	ELSIF ENABLE THEN
		IF trig_tmp OR trig_stored THEN (* manueller, automatischer oder externer Trigger *)
			trig_stored := FALSE;
			X.ADD_COM := 03; (* ADD DATA *)
			SAVE_DATA.TRIG_CNT := SAVE_DATA.TRIG_CNT + UDINT#1;
			SAVE_DATA.TRIG_CNT_TOTAL  := SAVE_DATA.TRIG_CNT_TOTAL + UDINT#1;
			(* ---------------- Debug-Message -----------------------*)
			(*IF _debug_enable THEN
				LOG_CL.NEW_MSG := 'FILE_XML1 - Trig: [~2]';
				LOG_CL.PRINTF[2] := DT_TO_STRING(DTI);
				LOG_MSG();
			END_IF;*)
			(* -----------------------------------------------------------------*)
		ELSE
			X.ADD_COM := 04;	(* ADD DATA REQ *)
		END_IF;
	END_IF;

END_CASE;
X.ADD_DATA_REQ := FALSE; (* externe Anforderung rücksetzen *)

(* ##################################### *)

CASE step_2 OF

00:	aw_ton(IN:= idx > 0 AND aw_enable , PT:= AUTO_CLOSE); (* AutoWrite Timer *)
	IF aw_ton.Q THEN (* Zeitgesteuertes Datenschreiben *)
		aw_aktiv := TRUE;
		step_2 := 10; (* Daten schreiben *)
		(* ---------------- Debug-Message -----------------------*)
		(*IF _debug_enable THEN
			LOG_CL.NEW_MSG := 'FILE_XML2 - AutoWrite: [~2]';
			LOG_CL.PRINTF[2] := DT_TO_STRING(DTI);
			LOG_MSG();
		END_IF;*)
		(* -----------------------------------------------------------------*)

	ELSIF idx + 256 > SIZEOF(PT.BUFFER) THEN (* Platz für Element vorhanden ? *)
		step_2 := 10; (* Daten schreiben *)
	ELSE
		wd_ton(IN:= FALSE, PT:= wd_time);
		wd_ton(IN:= TRUE);
		WHILE X.UCB.BUF_COUNT > 0 AND step_2 = 0 AND wd_ton.Q = FALSE DO

			X.UCB.D_MODE := 10;
			UCB(DATA:=X.UCB); (* Element lesen , aber noch nicht entfernen *)

			IF X.UCB.D_HEAD > WORD#16#F000 THEN (* F301 oder F201 *)
				X.UCB.D_MODE := 11;
				UCB(DATA:=X.UCB); (* Element entfernen *)

				FSD.MODE := WORD_TO_BYTE(SHR(SHL(X.UCB.D_HEAD,4),12)); (* 0X00 -> 000X = 3 create + write / 2 open + write *)
				FSD.OFFSET := UDINT#0; (* Start bei Dateianfang *)
				FSD.FILENAME := X.UCB.D_STRING; (* Dateiname *)
				PT.SIZE := UINT#0;
				SAVE_DATA.FN_REM := FSD.FILENAME; (* aktuellen Dateinamen remanent sichern *)

				IF FSD.MODE = BYTE#3 THEN	(* Datei neu anlegen -> dann zähler reset *)
					SAVE_DATA.TRIG_CNT := UDINT#0;
				END_IF;

				X.NEW_FILE := FSD.FILENAME;
				X.NEW_FILE_SIZE := UDINT#0;
				X.NEW_FILE_RTRIG := FALSE;
				step_2 := 20;

				(* Headerdaten schreiben *)
				IF FSD.MODE = BYTE#3 THEN
					str := '<?xml version="1.0" encoding="UTF-8"?><table>';
					_STRING_TO_BUFFER(STR:=str, POS:=idx, PT:=ADR(PT.BUFFER), SIZE:=SIZEOF(PT.BUFFER));
					idx := LEN(str);
					X.NEW_FILE_SIZE := total_bytes + INT_TO_UDINT(idx);
				END_IF;

				(* ---------------- Debug-Message -----------------------*)
				(*IF _debug_enable THEN
					LOG_CL.NEW_MSG := 'FILE_XML2 - Create: Mode [~1] , [~2]';
					LOG_CL.PRINTF[2] := DT_TO_STRING(DTI);
					LOG_CL.PRINTF[1] := BYTE_TO_STRING(FSD.MODE);
					LOG_MSG();
				END_IF;*)
				(* -----------------------------------------------------------------*)

			ELSIF X.UCB.D_HEAD = WORD#16#EE00 THEN (* LOG_STOP Command *)
				X.UCB.D_MODE := 11;
				UCB(DATA:=X.UCB); (* Element entfernen *)

				str := '</table>';
				_STRING_TO_BUFFER(STR:=str, POS:=idx, PT:=ADR(PT.BUFFER), SIZE:=SIZEOF(PT.BUFFER));
				idx := idx + LEN(str);
				log_stop := TRUE;
				step_2 := 10; (* Daten schreiben *)

			ELSE
				X.UCB.D_MODE := 11;
				UCB(DATA:=X.UCB); (* Element entfernen *)
				(* ---------------- Debug-Message -----------------------*)
				(*IF _debug_enable THEN
					LOG_CL.NEW_MSG := 'FILE_XML2 - BUF: TXT [~1],Pos [~2], [~3]';
					LOG_CL.PRINTF[1] := X.UCB.D_STRING;
					LOG_CL.PRINTF[2] := INT_TO_STRING(idx);
					LOG_CL.PRINTF[3] := DT_TO_STRING(DTI);
					LOG_MSG();
				END_IF;*)
				(* -----------------------------------------------------------------*)

				IF log_state = USINT#0 THEN
					str := '<row><entry>';
				ELSE
					str := '<entry>';
				END_IF;

				_STRING_TO_BUFFER(STR:=str, POS:=idx, PT:=ADR(PT.BUFFER), SIZE:=SIZEOF(PT.BUFFER));
				idx := idx + LEN(str);
				log_state := log_state + USINT#1;

				_STRING_TO_BUFFER(STR:=X.UCB.D_STRING, POS:=idx, PT:=ADR(PT.BUFFER), SIZE:=SIZEOF(PT.BUFFER));
				idx := idx + LEN(X.UCB.D_STRING);

				n := n + USINT#1;
				IF n >= X.ID_MAX THEN
					n := USINT#0;
					str := '</entry></row>';
					log_state := USINT#0;
				ELSE
					str := '</entry>';
				END_IF;
				_STRING_TO_BUFFER(STR:=str, POS:=idx, PT:=ADR(PT.BUFFER), SIZE:=SIZEOF(PT.BUFFER));
				idx := idx + LEN(str);
				X.NEW_FILE_SIZE := total_bytes + INT_TO_UDINT(idx);
			END_IF;
			wd_ton();
		END_WHILE;
	END_IF;

10:	IF idx > 0 THEN (* Daten schreiben *)
		FSD.MODE := BYTE#2; (* File_Open_Exist + File_Write *)
		FSD.OFFSET := UDINT#4294967294; (* 16#FFFF_FFFE ->Spezialcode: Daten automatisch an Dateiende anhängen *)
		PT.SIZE := INT_TO_UINT(idx); (* Datenlänge eintragen *)
		idx := 0;
		(* ---------------- Debug-Message -----------------------*)
		(*IF _debug_enable THEN
			LOG_CL.NEW_MSG := 'FILE_XML2 - WriteData: Mode [~3] Size [~1] , [~2]';
			LOG_CL.PRINTF[1] := UINT_TO_STRING(PT.SIZE);
			LOG_CL.PRINTF[2] := DT_TO_STRING(DTI);
			LOG_CL.PRINTF[3] := BYTE_TO_STRING(FSD.MODE);
			LOG_MSG();
		END_IF;*)
		(* -----------------------------------------------------------------*)
	END_IF;
	step_2 := 20;

20:	IF FSD.MODE = BYTE#0 THEN
		total_bytes := FSD.FILE_SIZE;
		X.NEW_FILE_SIZE := total_bytes + INT_TO_UDINT(idx);
		IF log_stop OR aw_aktiv THEN
			aw_aktiv := FALSE;
			FSD.MODE := BYTE#5; (* Datei schliessen *)
			(* ---------------- Debug-Message -----------------------*)
			(*IF _debug_enable THEN
				LOG_CL.NEW_MSG := 'FILE_XML2 - Close: [~2]';
				LOG_CL.PRINTF[2] := DT_TO_STRING(DTI);
				LOG_MSG();
			END_IF;*)
			(* -----------------------------------------------------------------*)
		END_IF;
		step_2 := 30;
	END_IF;

30:	IF FSD.MODE = BYTE#0 THEN (* Datei schliessen beendet *)
		IF log_stop THEN
			X.NEW_FILE_RTRIG := TRUE;
			log_stop := FALSE;
			SAVE_DATA.FN_REM := ''; (* remanenten Dateinamen löschen *)
		END_IF;
		step_2 := 00;
	END_IF;

END_CASE;

FS(FSD:=FSD,PT:=PT); (* FILE_SERVER *)
ERROR_C := BYTE_TO_DWORD(FSD.ERROR);
ERROR_T := SEL(FSD.ERROR > BYTE#0,BYTE#0,BYTE#1);

X.NEW_FILE_SIZE := total_bytes + INT_TO_UDINT(idx);
trig_m_last := TRIG_M;

(* revision history
ks	25. july. 2011	rev 1.0
	original version

ks	16. apr. 2012	rev 1.1
	neuer überarbeiteter Code für automatisches File-open/close
*)
END_FUNCTION_BLOCK

(* POU DLOG_MYSQL_DEMO, CFC *)
PROGRAM DLOG_MYSQL_DEMO
VAR
	cur_dt: DT;
	enable: BOOL := TRUE;
	trig_t : TIME := T#5s;
	trig_m : BOOL;
	error_c: DWORD;
	error_t: BYTE;

	x1 : DLOG_DT;
	x2 : DLOG_REAL;
	x3 : DLOG_DINT;
	x4 : DLOG_BOOL;
	x5 : DLOG_STRING;
	x : DLOG_DATA;
	mysql_info : MYSQL_INFO;

	RTC_2 : RTC_2;
	GEN_SIN_1: GEN_SIN;
	COUNT_DR : COUNT_DR;

	DLOG_STORE_MYSQL : DLOG_STORE_MYSQL;
	(*url : STRING := 'myuser:mypassword@127.0.0.1';*)
	url : STRING(STRING_LENGTH) := 'myuser:mypassword@192.168.178.21';
	db_name : STRING(64) := 'oscat_db';
	tb_name : STRING(64) := 'oscat_tb';
	auto_delete : UDINT := 0;
	timeout : TIME := t#10s;

END_VAR
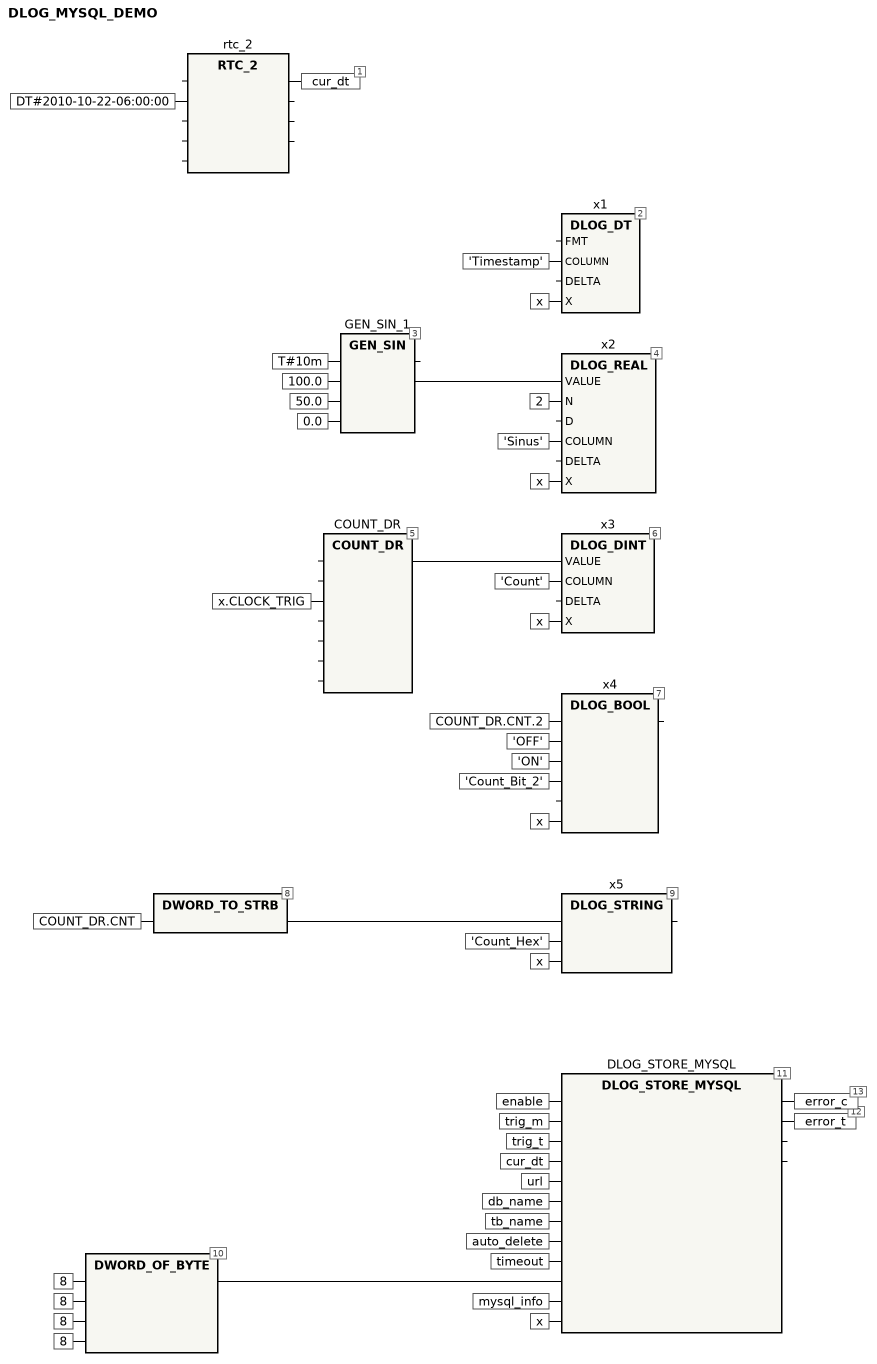
_CFC_ (* Continuous Function Chart, elements in execution order *)
#0 rtc_2:RTC_2(-, DT#2010-10-22-06:00:00, -, -, -)
#1 cur_dt <= #0.out 1
#2 x1:DLOG_DT(FMT: -, COLUMN: 'Timestamp', DELTA: -, X: x)
#3 GEN_SIN_1:GEN_SIN(T#10m, 100.0, 50.0, 0.0)
#4 x2:DLOG_REAL(VALUE: #3.out 2, N: 2, D: -, COLUMN: 'Sinus', DELTA: -, X: x)
#5 COUNT_DR:COUNT_DR(-, -, x.CLOCK_TRIG, -, -, -, -)
#6 x3:DLOG_DINT(VALUE: #5, COLUMN: 'Count', DELTA: -, X: x)
#7 x4:DLOG_BOOL(COUNT_DR.CNT.2, 'OFF', 'ON', 'Count_Bit_2', -, x)
#8 DWORD_TO_STRB(COUNT_DR.CNT)
#9 x5:DLOG_STRING(#8, 'Count_Hex', x)
#10 DWORD_OF_BYTE(8, 8, 8, 8)
#11 DLOG_STORE_MYSQL:DLOG_STORE_MYSQL(enable, trig_m, trig_t, cur_dt, url, db_name, tb_name, auto_delete, timeout, #10, mysql_info, x)
#12 error_t <= #11.out 2
#13 error_c <= #11.out 1
_END_CFC_
END_PROGRAM

(* POU DLOG_STORE_MYSQL, ST *)
FUNCTION_BLOCK DLOG_STORE_MYSQL
VAR_IN_OUT
	SQL_INFO : MYSQL_INFO;
	X : DLOG_DATA;
END_VAR
VAR_INPUT
	ENABLE : BOOL;
	TRIG_M : BOOL;
	TRIG_T : TIME;
	DTI : DT;
	URL : STRING(STRING_LENGTH);
	DB_NAME : STRING(64);
	TB_NAME : STRING(64);
	AUTO_DELETE : UDINT;
	TIMEOUT : TIME;
	DNS_IP4 : DWORD;
END_VAR
VAR_OUTPUT
	ERROR_C : DWORD;
	ERROR_T : BYTE;
END_VAR
VAR
	UCB : UNI_CIRCULAR_BUFFER;
	MYSQL_CONTROL: MYSQL_CONTROL;
	trig_auto : BOOL;
	trig_tmp : BOOL;
	trig_m_last : BOOL;
	dti_last : DT := DT#2070-02-06-06:28:15;
	enable_last : BOOL;
	step : INT;
	idx : INT;
	n : USINT;
	snd_text : STRING(STRING_LENGTH);
	snd_size : INT;
	sql_command : BYTE;
	next_step : INT;
	i1 : INT;
	i2 : INT;
	com: MYSQL_COM;
	del_dt : UDINT;
	del_start : BOOL;
	run : BOOL;

	(*
	LOG_MSG : LOG_MSG;
	_debug_enable : BOOL := TRUE;
	*)
END_VAR

(*
version 1.0		20. apr. 2012
programmer		ks
tested by		ks

DLOG_STORE_MYSQL der Baustein schreibt die DLOG Parameter in eine MySQL Datenbank
*)
X.DTI := DTI; (* Datum / Zeit eintragen *)
X.CLOCK_TRIG := DTI <> dti_last;
dti_last := DTI;
trig_auto := FALSE;
IF X.CLOCK_TRIG THEN (* Impuls in jeder Sekunde *)
	del_start := DT_TO_UDINT(DTI) - del_dt > AUTO_DELETE AND AUTO_DELETE > UDINT#0;
	IF TRIG_T >= T#1000ms THEN (* automatischer Trigger *)
		trig_auto := DT_TO_UDINT(DTI) MOD (TIME_TO_UDINT(TRIG_T) / UDINT#1000) = UDINT#0;
	END_IF;
END_IF;
X.ADD_COM := 00;

CASE step OF

00:	IF ENABLE AND enable_last = FALSE THEN
		COM.SQL_URL := URL;
		COM.TIMEOUT := TIMEOUT;
		COM.DNS_IP4 := DNS_IP4;
		COM.SQL_CON := TRUE;

		X.UCB.D_MODE := 99; (* Buffer reset - Alles löschen *)
		UCB(DATA:=X.UCB);

		X.ID_MAX := USINT#00;
		X.STORE_TYPE := BYTE#5; (* MySQL-Modus *)
		X.ADD_COM := 01; (* ADD INFO *)

		step := 05;
	END_IF;

05:	X.ADD_COM := 02; (* ADD HEADER *)
	step := 10;

10:	IF SQL_INFO.SQL_CONNECTED THEN
		sql_command := BYTE#3; (* CREATE DATABASE IF NOT EXISTS `db_name` *)
		snd_text :=  CONCAT('CREATE DATABASE IF NOT EXISTS `' ,DB_NAME);
		snd_text :=  CONCAT(snd_text, '`');
		next_step := 20;
	END_IF;

20:	sql_command := BYTE#2; (* 0x02 COM_INIT_DB mysql_select_db *)
	snd_text := DB_NAME;
	next_step := 30;

30:	(* CREATE TABLE IF NOT EXISTS tb_name (Timestamp TIMESTAMP NULL DEFAULT CURRENT_TIMESTAMP, n1,n2) *)
	sql_command := BYTE#0;
	idx := 5;
	n := USINT#0;
	WHILE sql_command = BYTE#0 DO
		IF n = USINT#0 THEN
			snd_text := CONCAT('CREATE TABLE IF NOT EXISTS `', TB_NAME);
			snd_text := CONCAT(snd_text,'` (`ID` BIGINT NOT NULL AUTO_INCREMENT PRIMARY KEY ,');
			snd_text := CONCAT(snd_text,' store_timestamp TIMESTAMP NULL DEFAULT CURRENT_TIMESTAMP');
		ELSIF n <= X.ID_MAX THEN
			X.UCB.D_MODE := 12; (* Element lesen und löschen *)
			UCB(DATA:=X.UCB);
			snd_text := CONCAT(', `',X.UCB.D_STRING);
			CASE WORD_TO_INT(SHR(X.UCB.D_HEAD,8)) OF
			02:	snd_text := CONCAT(snd_text, '` FLOAT'); (* REAL *)
			06:	snd_text := CONCAT(snd_text, '` BOOL'); (* BOOL *)
			08:	snd_text := CONCAT(snd_text, '` INT'); (* DINT *)
			13:	snd_text := CONCAT(snd_text, '` DATETIME'); (* DT *)
			ELSE
				snd_text := CONCAT(snd_text, '` VARCHAR(80)'); (* STRING(80) *)
			END_CASE;
		ELSE
			snd_text := ')';
			sql_command := BYTE#3;
			snd_size := idx + LEN(snd_text);
			next_step := 40;
		END_IF;
		_STRING_TO_BUFFER(str:=snd_text,pos:=idx,pt:=ADR(COM.S_BUF.BUFFER),size:=SIZEOF(COM.S_BUF.BUFFER)); (* String in puffer kopieren *)
		idx := idx + LEN(snd_text);
		n := n + USINT#1;

		(*####################  DEBUG-MESSAGE  ###################################*)
		(*IF _debug_enable THEN
			LOG_CL.NEW_MSG := 'dlog_mysql: create >~1<';
			LOG_CL.PRINTF[1] := snd_text;
			LOG_MSG();
		END_IF;*)
		(*########################################################################*)
	END_WHILE;

40:	IF del_start THEN
		del_start := FALSE;
		sql_command := BYTE#3; (* DELETE FROM `tb_name` WHERE TIMESTAMPDIFF(SECOND, Timestamp, NOW()) > xxx *)
		snd_text := CONCAT('DELETE FROM `', TB_NAME);
		snd_text := CONCAT(snd_text, '` WHERE TIMESTAMPDIFF(SECOND, store_timestamp, NOW()) > ');
		snd_text := CONCAT(snd_text, UDINT_TO_STRING(AUTO_DELETE));
		next_step := 40;
		del_dt := DT_TO_UDINT(DTI);
		(*####################  DEBUG-MESSAGE  ###################################*)
		(*IF _debug_enable THEN
			LOG_CL.NEW_MSG := 'dlog_mysql: # delete time:~1 >~2<';
			LOG_CL.PRINTF[1] := UDINT_TO_STRING(AUTO_DELETE);
			LOG_CL.PRINTF[2] := snd_text;
			LOG_MSG();
		END_IF;*)
		(*########################################################################*)

         (* INSERT INTO `tb_name` VALUES (CURRENT_TIMESTAMP,  "n1","n2") *)
	ELSIF X.UCB.BUF_COUNT >= USINT_TO_INT(X.ID_MAX) AND step > 0 THEN (* Neue Datenreihe(n) vorhanden *)
		idx := 5;
		n := USINT#0;
		sql_command := BYTE#0;
		WHILE sql_command = BYTE#0 DO
			IF n = USINT#0 THEN
				snd_text := CONCAT('INSERT INTO `', TB_NAME);
				snd_text := CONCAT(snd_text,'` VALUES (NULL, CURRENT_TIMESTAMP');
			ELSIF n <= X.ID_MAX THEN
				X.UCB.D_MODE := 12; (* Element lesen und löschen *)
				UCB(DATA:=X.UCB);
				snd_text := CONCAT(', "',X.UCB.D_STRING);
				snd_text := CONCAT(snd_text, '"');
			ELSE
				snd_text := ')';
				sql_command := BYTE#3;
				snd_size := idx + LEN(snd_text);
				next_step := 40;
			END_IF;
			_STRING_TO_BUFFER(str:=snd_text,pos:=idx,pt:=ADR(COM.S_BUF.BUFFER),size:=SIZEOF(COM.S_BUF.BUFFER)); (* String in puffer kopieren *)
			idx := idx + LEN(snd_text);
			n := n + USINT#1;

			(*####################  DEBUG-MESSAGE  ###################################*)
			(*IF _debug_enable THEN
				LOG_CL.NEW_MSG := 'dlog_mysql: insert >~1<';
				LOG_CL.PRINTF[1] := snd_text;
				LOG_MSG();
			END_IF;*)
			(*########################################################################*)
		END_WHILE;
	END_IF;

	IF ENABLE THEN 	(* LOG-Trigger verarbeiten *)
		trig_tmp := (TRIG_M AND NOT trig_m_last) OR trig_auto OR X.ADD_DATA_REQ;

		IF trig_tmp THEN (* manueller, automatischer oder externer Trigger *)
			X.ADD_COM := 03; (* ADD DATA *)
			(* ---------------- Debug-Message -----------------------*)
			(*IF _debug_enable THEN
				LOG_CL.NEW_MSG := 'dlog_mysql: Trigger: DATE [~2]';
				LOG_CL.PRINTF[2] := DT_TO_STRING(DTI);
				LOG_MSG();
			END_IF;*)
			(* -----------------------------------------------------------------*)
		ELSE
			X.ADD_COM := 04;	(* ADD DATA REQ *)
		END_IF;
	ELSE
		COM.SQL_CON := FALSE; (* MySQL Verbindung beenden *)
		step := 0;
	END_IF;

(* ~~~~~~~~~~~~~~~~~~~~~~ *)

199:IF COM.SQL_RCV_STATE = BYTE#1 THEN (* OK *)
		step := next_step;
	ELSIF COM.SQL_RCV_STATE = BYTE#2 THEN  (* FEHLER *)
		step := 0;
	END_IF;

END_CASE;

(* ########################## *)
(* SQL-Kommando ausführen *)
IF sql_command > BYTE#0 THEN
	IF snd_size > 0 THEN
		COM.S_BUF.SIZE := INT_TO_UINT(snd_size);
		snd_size := 0;
	ELSE
		_STRING_TO_BUFFER(str:=snd_text,pos:=5,pt:=ADR(COM.S_BUF.BUFFER),size:=SIZEOF(COM.S_BUF.BUFFER)); (* String in puffer kopieren *)
		COM.S_BUF.SIZE := INT_TO_UINT(5 + LEN(snd_text));
		snd_text := '';
	END_IF;

	i2 := UINT_TO_INT(COM.S_BUF.SIZE) - 1; (* alle " zeichen mit ' ersetzen *)
	FOR i1 := 5 TO i2 DO
		IF COM.S_BUF.BUFFER[i1] = BYTE#34 THEN
			COM.S_BUF.BUFFER[i1] := BYTE#39;
		END_IF;
	END_FOR;

	COM.S_BUF.BUFFER[4] := sql_command;
	COM.SQL_PACKET_NO := BYTE#255;
	sql_command := BYTE#0;
	step := 199;
END_IF;

(* ########################## *)

MYSQL_CONTROL(COM:= COM, INFO:=SQL_INFO);
ERROR_C := COM.ERROR_C;
ERROR_T := COM.ERROR_T;

IF COM.ERROR_T > BYTE#0 THEN  (* FEHLER *)
	step := 0;
END_IF;

(* ########################## *)

trig_m_last := TRIG_M;
enable_last := ENABLE;
run := step > 0;

(* revision history
ks	20. apr. 2012	rev 1.0
	original version

*)
END_FUNCTION_BLOCK

(* POU MYSQL_CONTROL, ST *)
FUNCTION_BLOCK MYSQL_CONTROL
VAR_IN_OUT
	COM : MYSQL_COM;
	INFO : MYSQL_INFO;
END_VAR
VAR_OUTPUT
END_VAR
VAR
	IP_C : IP_C;
	URL_DATA : url;
	DNS_CLIENT : DNS_CLIENT;
	IPC : IP_CONTROL;

	step : INT;
	snd_step : INT;
	TON_WAIT : TON;
	last_step : INT;
	idx1 : INT;
	idx2 : INT;
	idx3 : INT;
	dw_tmp : DWORD;
	timeout1 : TIME;
	timeout2 : TIME;
	ip_c_red_disable : BOOL;
	auth_password : STRING(64);
	auth_run : BOOL;
	MYSQL_AUTH : MYSQL_AUTH;
	scramble1_buffer : ARRAY [0..19] OF BYTE;
	scramble2_buffer : ARRAY [0..19] OF BYTE;
	charset_number : BYTE := 16#08;
	max_packet_size : DWORD := 1024;
	client_flags : DWORD := 16#0003_8601;

	(*
	LOG_MSG : LOG_MSG;
	_debug_enable : BOOL := TRUE;
	*)

END_VAR

(*
version 1.0		16. apr. 2012
programmer		ks
tested by		ks

MYSQL_CONTROL führt einen SQL Befehl auf einem MySQL-Server durch 
*)
CASE step OF

00:	IF COM.SQL_CON THEN
		timeout1 := MAX(T#10s,COM.TIMEOUT);
		timeout2 := timeout1 + T#1s;
		INFO.SQL_ERROR := '';
		COM.ERROR_C := DWORD#0;
		COM.ERROR_T := BYTE#0;
		URL_DATA := STRING_TO_URL(STR:=COM.SQL_URL,DEFAULT_PROTOCOL:='',DEFAULT_PATH:='/');
		step := 10;
	END_IF;

10:	IF DNS_CLIENT.DONE THEN
		step := 20;
	ELSIF DNS_CLIENT.ERROR <> DWORD#0 THEN
		COM.ERROR_C := DNS_CLIENT.ERROR;
		COM.ERROR_T := BYTE#1;
		step := 980;
	END_IF;

20:	(* MySQL Steuerkanal einrichten *)
	IF URL_DATA.PORT = WORD#0 THEN
		URL_DATA.PORT := WORD#3306; (* Standard Port *)
	END_IF;
	IP_C.C_PORT := URL_DATA.PORT; (* Portnummer eintragen *)
  	IP_C.C_IP := DNS_CLIENT.IP4; (* IP eintragen *)
  	IP_C.C_MODE := BYTE#0; (* Mode: TCP+ACTIV+PORT *)
  	IP_C.TIME_RESET := TRUE; (* Zeitueberwachung rücksetzen *)
  	IP_C.C_ENABLE := TRUE; (* Verbindungsaufbau freigeben *)
  	IP_C.R_OBSERVE := TRUE; (* Empfangsueberwachung *)
	COM.R_BUF.SIZE := UINT#0;
	COM.SQL_RCV_STATE := BYTE#0;
	step := 30;

30:	IF COM.SQL_RCV_STATE = BYTE#1 THEN
		INFO.SERVER_PROTOCOL_VERSION := COM.R_BUF.BUFFER[4];

		(* ende markierung von string server_version suchen *)
		idx2 := UINT_TO_INT(COM.R_BUF.SIZE) - 1;
		FOR idx1 := 5 TO idx2 DO
			IF COM.R_BUF.BUFFER[idx1] = BYTE#0 THEN EXIT; END_IF;
		END_FOR;
		idx1 := idx1 + 5; (* terminierung und thread-id überspringen *)

		FOR idx2:=0 TO 7 DO	(* Byte 0-7 *)
			scramble1_buffer[idx2] := COM.R_BUF.BUFFER[idx1];
			idx1 := idx1 + 1;
		END_FOR;
		idx1 := idx1 + 1;
		idx2 := idx1 + 1;
		INFO.SERVER_CAPABILITIES := WORD_OF_BYTE(COM.R_BUF.BUFFER[idx2], COM.R_BUF.BUFFER[idx1]);
		idx1 := idx1 + 2;
		INFO.SERVER_LANGUAGE := COM.R_BUF.BUFFER[idx1];
		idx1 := idx1 + 1;
		idx2 := idx1 + 1;
		INFO.SERVER_STATUS := WORD_OF_BYTE(COM.R_BUF.BUFFER[idx2], COM.R_BUF.BUFFER[idx1]);
		idx1 := idx1 + 15;

		FOR idx2:=8 TO 19 DO	(* Byte 8-19 *)
			scramble1_buffer[idx2] := COM.R_BUF.BUFFER[idx1];
			idx1 := idx1 + 1;
		END_FOR;

		IF INFO.SERVER_PROTOCOL_VERSION < BYTE#10 THEN  (* Error: protocol version zu niedrig *)
			COM.ERROR_T := BYTE#2;
			COM.ERROR_C := DWORD#1;
			step := 980;
		ELSIF URL_DATA.PASSWORD = '' THEN
			step := 50;
		ELSE
			auth_password := URL_DATA.PASSWORD;
			auth_run := TRUE;
			step := 40;
		END_IF;
	END_IF;

40:	MYSQL_AUTH(RUN:= auth_run,PASSWORD:= auth_password ,MESSAGE:= scramble1_buffer,SCRAMBLE:= scramble2_buffer);
	IF NOT auth_run THEN
		step := 50;
	END_IF;

50: (* Client Authentication Packet *)
	(* Byte 0-3 werden später eingetragen *)
	COM.S_BUF.BUFFER[04] := BYTE_OF_DWORD(client_flags, BYTE#0); (* client_flags *)
	COM.S_BUF.BUFFER[05] := BYTE_OF_DWORD(client_flags, BYTE#1);
	COM.S_BUF.BUFFER[06] := BYTE_OF_DWORD(client_flags, BYTE#2);
	COM.S_BUF.BUFFER[07] := BYTE_OF_DWORD(client_flags, BYTE#3);
	COM.S_BUF.BUFFER[08] := BYTE_OF_DWORD(max_packet_size, BYTE#0); (* max_packet_size *)
	COM.S_BUF.BUFFER[09] := BYTE_OF_DWORD(max_packet_size, BYTE#1);
	COM.S_BUF.BUFFER[10] := BYTE_OF_DWORD(max_packet_size, BYTE#2);
	COM.S_BUF.BUFFER[11] := BYTE_OF_DWORD(max_packet_size, BYTE#3);
	COM.S_BUF.BUFFER[12] := charset_number; (* charset_number *)
	FOR idx1 := 13 TO 35 DO (* 23 bytes filler always 0x00.. *)
		COM.S_BUF.BUFFER[idx1] := BYTE#0;
	END_FOR;
	idx3 := LEN(URL_DATA.USER);
	FOR idx2 :=1 TO idx3 DO
		COM.S_BUF.BUFFER[idx1] := CODE(URL_DATA.USER, idx2);
		idx1 := idx1 + 1;
	END_FOR;
	COM.S_BUF.BUFFER[idx1] := BYTE#0; (* String terminierung eintragen *)
	idx1 := idx1 + 1;
	IF LEN(URL_DATA.PASSWORD) = 0 THEN
		COM.S_BUF.BUFFER[idx1] := BYTE#0; (* scramble_buff length *)
	ELSE
		COM.S_BUF.BUFFER[idx1] := BYTE#20; (* scramble_buff length *)
		FOR idx2 :=0 TO 19 DO
			idx1 := idx1 + 1;
			COM.S_BUF.BUFFER[idx1] := scramble2_buffer[idx2];
		END_FOR;
	END_IF;
	COM.S_BUF.SIZE  := INT_TO_UINT(idx1 + 1); (* Sendelänge eintragen *)

	step := 60;

60:	IF COM.SQL_RCV_STATE = BYTE#1 THEN
		INFO.SQL_CONNECTED := TRUE;
		step := 300;
	END_IF;

(* ================================================== *)

300:	step := SEL(COM.SQL_CON,700,310); (* Schritt-Selektion *)

310:	step := 300; (* dummy step *)

(* ================================================== *)

700: (* COM_QUIT *)
	COM.S_BUF.BUFFER[04] := BYTE#1; (* 0x01 COM_QUIT mysql_close *)
	COM.S_BUF.SIZE := UINT#5; (* Sendelänge eintragen *)
	COM.SQL_PACKET_NO := BYTE#255;
	ip_c_red_disable := TRUE;
	step := 710;

710:	IF IP_C.C_STATE = BYTE#0 THEN (* Verbindung durch SQL-Server beendet ? *)
		step := 980;
	END_IF;

(* ================================================== *)

980:IP_C.C_ENABLE := FALSE; (* MYSQL Steuerkanal schliessen *)
	ip_c_red_disable := FALSE;
	INFO.SQL_CONNECTED := FALSE;
	COM.SQL_CON := FALSE;
	COM.S_BUF.SIZE := UINT#0;
	COM.R_BUF.SIZE := UINT#0;
	snd_step := 0;
	step := 990;
	(*####################  DEBUG-MESSAGE  ###################################*)
	(*IF _debug_enable THEN
		LOG_CL.NEW_MSG := 'QUIT: ERROR CODE >~1< TYPE >~2<';
		LOG_CL.PRINTF[1] := DWORD_TO_STRH(COM.ERROR_C);
		LOG_CL.PRINTF[2] := BYTE_TO_STRING(COM.ERROR_T);
		LOG_MSG();
	END_IF;*)
	(*########################################################################*)

990:IF IP_C.C_STATE = BYTE#0 THEN
		step := 0;
	END_IF;

END_CASE;

(* ++++++++++++++++++++++++++++++++++++++++++++++++++++++++++ *)

IF step >= 30 THEN
	IF COM.R_BUF.SIZE >= UINT#3 AND COM.SQL_RCV_STATE = BYTE#0 THEN (* Daten wurden empfangen ? *)
		IF DWORD_TO_UINT(DWORD_OF_BYTE(BYTE#0, COM.R_BUF.BUFFER[2], COM.R_BUF.BUFFER[1], COM.R_BUF.BUFFER[0])) + UINT#4 = COM.R_BUF.SIZE THEN
			COM.SQL_PACKET_NO := COM.R_BUF.BUFFER[3];
			IF COM.R_BUF.BUFFER[4] = BYTE#16#FF THEN
				idx2 := 13; (* Error String - Erstes Zeichen *)
				idx3 := UINT_TO_INT(COM.R_BUF.SIZE) - 1; (* Error String - Letztes Zeichen *)
				FOR idx1 := idx2 TO idx3 DO (* alle ' durch ´ ersetzen *)
					IF COM.R_BUF.BUFFER[idx1] = BYTE#39 THEN
						COM.R_BUF.BUFFER[idx1] := BYTE#96;
					END_IF;
				END_FOR;
				INFO.SQL_ERROR := BUFFER_TO_STRING(PT:=ADR(COM.R_BUF.BUFFER),SIZE:=COM.R_BUF.SIZE,START:=INT_TO_UINT(idx2),STOP:=INT_TO_UINT(idx3));
				COM.ERROR_T := BYTE#3;
				COM.ERROR_C := DWORD_OF_BYTE(BYTE#0,BYTE#0,COM.R_BUF.BUFFER[6], COM.R_BUF.BUFFER[5]);
				COM.SQL_RCV_STATE := BYTE#2;
				COM.R_BUF.SIZE := UINT#0; (* Empfangsbuffer nach Fehler rücksetzen *)
				step := 980;
			ELSE
				COM.SQL_RCV_STATE := BYTE#1;
				IP_C.R_OBSERVE := FALSE;

				(*####################  DEBUG-MESSAGE  ###################################*)
				(*IF _debug_enable THEN
					LOG_CL.NEW_MSG := 'RCV: size >~1<';
					LOG_CL.PRINTF[1] := UINT_TO_STRING(COM.R_BUF.SIZE);
					LOG_MSG();
				END_IF;*)
				(*########################################################################*)
			END_IF;
		END_IF;
	END_IF;
END_IF;

(* automatisches Datensenden *)

CASE snd_step OF

00:	IF COM.S_BUF.SIZE > UINT#0 THEN
		dw_tmp := UINT_TO_DWORD(COM.S_BUF.SIZE - UINT#4); (* packet_length *)
		COM.S_BUF.BUFFER[0] := BYTE_OF_DWORD(dw_tmp, BYTE#0);
		COM.S_BUF.BUFFER[1] := BYTE_OF_DWORD(dw_tmp, BYTE#1);
		COM.S_BUF.BUFFER[2] := 0;
		COM.SQL_PACKET_NO := COM.SQL_PACKET_NO + 1;
		COM.S_BUF.BUFFER[3] := COM.SQL_PACKET_NO;

		IP_C.R_OBSERVE := TRUE;
		COM.R_BUF.SIZE := UINT#0; (* Empfangsbuffer rücksetzen *)
		COM.SQL_RCV_STATE := BYTE#0;

	        (*####################  DEBUG-MESSAGE  ###################################*)
	        (*IF _debug_enable THEN
	          LOG_CL.NEW_MSG := 'SND: size >~1<';
	          LOG_CL.PRINTF[1] := UINT_TO_STRING(COM.S_BUF.SIZE);
	          LOG_MSG();
	        END_IF;*)
	        (*########################################################################*)

		snd_step := 10;
	END_IF;

10:	IF COM.S_BUF.SIZE = UINT#0 THEN (* warten bis alle daten gesendet sind *)
		snd_step := 0;
	END_IF;

END_CASE;

(* Globale Fehlerbehandlung für Haupt-Routine *)
IF COM.ERROR_T = BYTE#0 AND step > 20 THEN (* noch kein Fehler gespeichert und Hauptroutine aktiv *)
	IF IP_C.ERROR > DWORD#0 AND IP_C.C_ENABLE AND NOT IP_C.TIME_RESET THEN  (* IP Control *)
		IF ip_c_red_disable = FALSE OR IP_C.ERROR <> DWORD#16#FD000000 THEN
			COM.ERROR_C := IP_C.ERROR;
			COM.ERROR_T := BYTE#2;
			step := 980;
		END_IF;
	END_IF;
END_IF;

IF TON_WAIT.Q THEN (* Ablaufstörung - Schrittkette *)
	COM.ERROR_C := INT_TO_DWORD(step); (* aktuellen Schritt eintragen *)
	COM.ERROR_T := BYTE#5;
	step := 980;
END_IF;

(* ######################################################## *)

DNS_CLIENT(IP_C:=IP_C, S_BUF:=COM.S_BUF, R_BUF:=COM.R_BUF, DOMAIN:=URL_DATA.DOMAIN, IP4_DNS:= COM.DNS_IP4, ACTIVATE:=step=10); (* DNS-Client *)
IPC(IP:= DWORD#0, PORT:= WORD#0 , TIME_OUT:= timeout1, IP_C:= IP_C, S_BUF:= COM.S_BUF, R_BUF:= COM.R_BUF); (* MYSQL Steuerkanal *)

TON_WAIT(IN:=step = last_step AND step > 0,PT:=timeout2);
last_step := step;

(* revision history
ks	20. apr. 2012	rev 1.0
	original version

*)
END_FUNCTION_BLOCK

(* POU MYSQL_AUTH, ST *)
FUNCTION_BLOCK MYSQL_AUTH
VAR_IN_OUT
	RUN : BOOL;
	PASSWORD : STRING(64);
	MESSAGE : ARRAY [0..19] OF BYTE;
	SCRAMBLE : ARRAY [0..19] OF BYTE;
END_VAR
VAR
	SHA1_STREAM : SHA1_STREAM;
	buf : ARRAY [0..63] OF BYTE;
	sha_mode : INT;
	step : INT;
	size : UDINT;
	pos : UDINT;
	i : INT;
	i2: INT;
	scramble1 : ARRAY [0..19] OF BYTE;
	scramble2 : ARRAY [0..19] OF BYTE;
END_VAR

(*
version 1.0		16. apr. 2012
programmer		ks
tested by		ks

MYSQL_AUTH führt das Passwort-Hashing fuer die Anmeldung bei einem MySQL 4.1 Server durch 
*)
IF NOT RUN THEN RETURN; END_IF;
CASE step OF

0:	CASE sha_mode OF
	0:	sha_mode := 1; (* Initialisierung *)
		size := INT_TO_UDINT(LEN(PASSWORD));
		i2 := UDINT_TO_INT(size) - 1;
		FOR i := 0 TO 63 DO
			IF i <= i2 THEN
				buf[i] := CODE(STR:=PASSWORD,POS:=i+1);
			ELSE
				buf[i] := BYTE#0;
			END_IF;
		END_FOR;

	3:	scramble1 := SCRAMBLE;
		sha_mode := 1; (* Initialisierung *)
		size := UDINT#20;
		FOR i := 0 TO 19 DO
			buf[i] := scramble1[i];
		END_FOR;
		step := 10;
	END_CASE;

10:	IF sha_mode = 3 THEN
		sha_mode := 1; (* Initialisierung *)
		scramble2 := SCRAMBLE;
		size := UDINT#40;
		FOR i := 0 TO 19 DO
			buf[i] := message[i];
			buf[i+20] := scramble2[i];
		END_FOR;
		step :=20;
	END_IF;

20:	IF sha_mode = 3 THEN
		sha_mode := 0; (* Stop *)
		FOR i:= 0 TO 19 DO
			SCRAMBLE[i] := SCRAMBLE[i] XOR scramble1[i];
		END_FOR;
		step :=0;
		RUN := FALSE;
	END_IF;
END_CASE;

SHA1_STREAM(SIZE:=size, MODE:=sha_mode, BUF:=buf, SHA1:=SCRAMBLE, POS=>pos);

(* revision history
ks	20. apr. 2012	rev 1.0
	original version

*)
END_FUNCTION_BLOCK

(* POU SHA1_STREAM, ST *)
FUNCTION_BLOCK SHA1_STREAM
VAR_IN_OUT
	MODE : INT;
	BUF : ARRAY [0..63] OF BYTE;
	SHA1 : ARRAY [0..19] OF BYTE;
	SIZE : UDINT;
END_VAR

VAR_OUTPUT
	POS : UDINT;
END_VAR

VAR
	hash : ARRAY [0..4] OF DWORD;
	end : UDINT;
	block : UDINT;
	pad_1 : BOOL;
	w : ARRAY [0..79] OF DWORD;
	n : INT;
	n1 : INT;
	a : DWORD;
	b : DWORD;
	c : DWORD;
	d : DWORD;
	e : DWORD;
	f : DWORD;
	k : DWORD;
	x : DWORD;
	z : INT;
END_VAR

(*
version 1.0	06. dec. 2009
programmer 	ks
tested BY	ks

SHA1_STREAM berechnet den SHA1 Hash eines Datenstromes
*)
CASE MODE OF

1:	(* Initialisierung der Hash-Werte *)
	hash[0] := DWORD#16#67452301;
	hash[1] := DWORD#16#EFCDAB89;
	hash[2] := DWORD#16#98BADCFE;
	hash[3] := DWORD#16#10325476;
	hash[4] := DWORD#16#C3D2E1F0;

	(* Buffer initialisieren *)
	FOR n := 16 TO 79 DO
   		w[n] := DWORD#0;
	END_FOR;

	block := SHR(SIZE,6) + BOOL_TO_UDINT((UDINT_TO_BYTE(SIZE) AND 16#3F) > 55);	(* benötigte Blocks errechnen *)

	pad_1 := FALSE;
	POS := 0;
	End := SIZE;
	SIZE := MIN(64,End);
	MODE := 2;

2:	FOR n := UDINT_TO_INT(SIZE) TO 63 DO (* Fuell-Bytes anhängen *)
		BUF[n] := 0;
	END_FOR;

	IF SIZE < 64 AND NOT pad_1 THEN
		BUF[SIZE] := 2#1000_0000;
		pad_1 := TRUE;
	END_IF;

	POS := POS + SIZE;
	SIZE := MIN(64,End - POS);

	n := 0;	(* Byte-Array in DWORD-Array umkopieren *)
	FOR n1 := 0 TO 15 DO
		w[n1] := DWORD_OF_BYTE(BUF[n],BUF[n+1],BUF[n+2],BUF[n+3]);
		n := n + 4;
	END_FOR;

	IF block = 0 THEN (* am Ende des letzten Blocks die Datenlänge eintragen *)
		w[15] := SHL(UDINT_TO_DWORD(End),3); (* Anzahl Datenbits eintragen *)
		MODE := 3;
	ELSE
		block := block - 1;
	END_IF;

	FOR n := 16 TO 79 DO (* erweitern der 16 32-bit-Worte auf 80 32-bit-Worte *)
		w[n] := ROL(w[n-3] XOR w[n-8] XOR w[n-14] XOR w[n-16],1);
	END_FOR;

	a := hash[0];
	b := hash[1];
	c := hash[2];
	d := hash[3];
	e := hash[4];

	FOR n := 0 TO 79 DO
		IF n <= 19 THEN
			f := (b AND c) OR (NOT(b) AND d);
			k := DWORD#16#5A827999;
		ELSIF n <= 39 THEN
			f := b XOR c XOR d;
			k := DWORD#16#6ED9EBA1;
		ELSIF n <= 59 THEN
			f := (b AND c) OR (b AND d) OR (c AND d);
			k := DWORD#16#8F1BBCDC;
		ELSE
			f := b XOR c XOR d;
			k := DWORD#16#CA62C1D6;
		END_IF;

		x := ROL(a,5) + f + e + k + w[n];
		e := d;
		d := c;
		c := ROL(b,30);
		b := a;
		a := x;
	END_FOR;

	(* aktuelle Hash-Werte zum letzten Wert addieren *)
	hash[0] := hash[0] + a;
	hash[1] := hash[1] + b;
	hash[2] := hash[2] + c;
	hash[3] := hash[3] + d;
	hash[4] := hash[4] + e;

END_CASE;

IF MODE = 3 THEN
	z := 0;
	FOR n := 0 TO 4 DO (* konvertiere DWORD auf BYTE-Array *)
		FOR n1 := 0 TO 3 DO
			hash[n] := ROL(hash[n],8);
			SHA1[z] := DWORD_TO_BYTE(hash[n]);
			z := z + 1;
		END_FOR;
	END_FOR;
END_IF;

(* revision history

ks	6. dec. 2009 rev 1.0
	original version

*)
END_FUNCTION_BLOCK

(* POU DLOG_RRD_DEMO, CFC *)
PROGRAM DLOG_RRD_DEMO
VAR
	cur_dt: DT;
	trig_t : TIME := T#50s;
	trig_m : BOOL;

	rrd_error_c : DWORD;
	rrd_error_t : BYTE;
	rrd_enable : BOOL := TRUE;
	(*rrd_url : STRING(STRING_LENGTH) := 'http://xxx.com/myhouse/rrd/test_rrd.php?rrd_db=test.rrd&value=';*)
	rrd_url : STRING(STRING_LENGTH) := '192.168.178.21/rrd/test_rrd2.php?rrd_db=test.rrd&value=';
	rrd_timeout: TIME := t#5s;

	RTC_2 : RTC_2;
	DLOG_STORE_RRD : DLOG_STORE_RRD;

	x : DLOG_DATA;
	x1 : DLOG_DINT;
	x2 : DLOG_DINT;
	x3 : DLOG_REAL;
	x4 : DLOG_REAL;
	x5 : DLOG_REAL;
	x6 : DLOG_REAL;
	x7 : DLOG_REAL;

	GEN_SIN_1 : GEN_SIN;
	GEN_SIN_2 : GEN_SIN;
	GEN_SIN_3 : GEN_SIN;
	GEN_RMP_1: GEN_RMP;
	GEN_RMP_2: GEN_RMP;
END_VAR
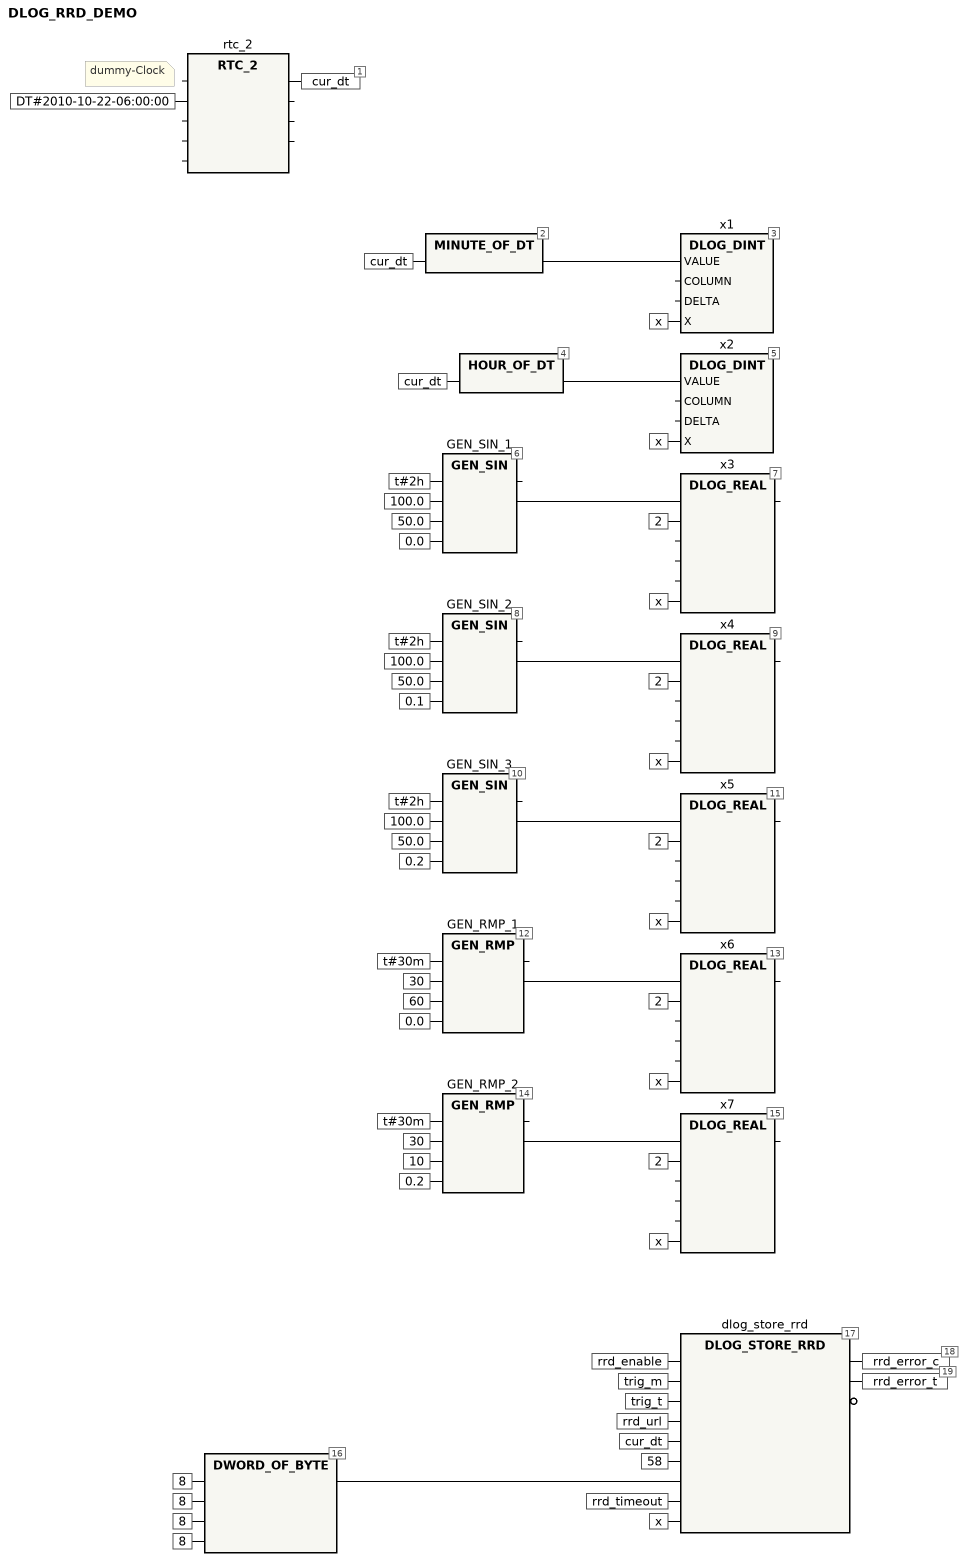
_CFC_ (* Continuous Function Chart, elements in execution order *)
#0 rtc_2:RTC_2(-, DT#2010-10-22-06:00:00, -, -, -)
#1 cur_dt <= #0.out 1
#2 MINUTE_OF_DT(cur_dt)
#3 x1:DLOG_DINT(VALUE: #2, COLUMN: -, DELTA: -, X: x)
#4 HOUR_OF_DT(cur_dt)
#5 x2:DLOG_DINT(VALUE: #4, COLUMN: -, DELTA: -, X: x)
#6 GEN_SIN_1:GEN_SIN(t#2h, 100.0, 50.0, 0.0)
#7 x3:DLOG_REAL(#6.out 2, 2, -, -, -, x)
#8 GEN_SIN_2:GEN_SIN(t#2h, 100.0, 50.0, 0.1)
#9 x4:DLOG_REAL(#8.out 2, 2, -, -, -, x)
#10 GEN_SIN_3:GEN_SIN(t#2h, 100.0, 50.0, 0.2)
#11 x5:DLOG_REAL(#10.out 2, 2, -, -, -, x)
#12 GEN_RMP_1:GEN_RMP(t#30m, 30, 60, 0.0)
#13 x6:DLOG_REAL(#12.out 2, 2, -, -, -, x)
#14 GEN_RMP_2:GEN_RMP(t#30m, 30, 10, 0.2)
#15 x7:DLOG_REAL(#14.out 2, 2, -, -, -, x)
#16 DWORD_OF_BYTE(8, 8, 8, 8)
#17 dlog_store_rrd:DLOG_STORE_RRD(rrd_enable, trig_m, trig_t, rrd_url, cur_dt, 58, #16, rrd_timeout, x)
#18 rrd_error_c <= #17.out 1
#19 rrd_error_t <= #17.out 2
(* dummy-Clock *)
_END_CFC_
END_PROGRAM

(* POU DLOG_STORE_RRD, ST *)
FUNCTION_BLOCK DLOG_STORE_RRD
VAR_IN_OUT
	X : DLOG_DATA;
END_VAR
VAR_INPUT
	ENABLE : BOOL;
	TRIG_M : BOOL;
	TRIG_T : TIME;
	URL : STRING(STRING_LENGTH);
	DTI : DT;
	SEP : BYTE;
	DNS_IP4 : DWORD;
	TIMEOUT : TIME;
END_VAR
VAR_OUTPUT
	ERROR_C : DWORD;
	ERROR_T : BYTE;
END_VAR
VAR
	UCB : UNI_CIRCULAR_BUFFER;
	IP_C : IP_C; (* IP_Control Verwaltungsstruktur *)
	S_BUF : NETWORK_BUFFER;
	R_BUF : NETWORK_BUFFER;
	URL_DATA : url;
	DNS_CLIENT : DNS_CLIENT;
	HTTP_GET : HTTP_GET;
	IPC : IP_CONTROL;

	trig_auto : BOOL;
	trig_stored : BOOL;
	trig_tmp : BOOL;
	trig_m_last : BOOL;
	dti_last : DT := DT#2070-02-06-06:28:15;
	step_1 : INT;
	step_2 : INT;
	sep_char : STRING(1);
	url_query : STRING(STRING_LENGTH);
	n : INT;

	(*
	LOG_MSG : LOG_MSG;
	_debug_enable : BOOL := TRUE;
	*)
END_VAR

(*
version 1.3		16. apr. 2012
programmer		ks
tested by			ks

DLOG_STORE_RRD der Baustein übergibt die DLOG Parameter an einen RoundRobinDatabase-Server
*)
X.DTI := DTI; (* Datum / Zeit eintragen *)
X.CLOCK_TRIG := DTI <> dti_last;
dti_last := DTI;
trig_auto := FALSE;
IF X.CLOCK_TRIG THEN (* Impuls in jeder Sekunde *)
	IF TRIG_T >= T#1000ms THEN (* automatischer Trigger *)
		trig_auto := DT_TO_UDINT(DTI) MOD (TIME_TO_UDINT(TRIG_T) / UDINT#1000) = UDINT#0;
	END_IF;
END_IF;

CASE step_1 OF

00:	IF ENABLE THEN
		X.ID_MAX := USINT#00;
		X.ADD_COM := 01; (* ADD INFO *)
		X.STORE_TYPE := BYTE#1; (* RRD-Modus *)

		ERROR_T := BYTE#0;
		ERROR_C := DWORD#0;

		X.UCB.D_MODE := 99;
		UCB(DATA:=X.UCB); (* Buffer löschen *)

		URL_DATA:=STRING_TO_URL(STR:=URL,DEFAULT_PROTOCOL:='',DEFAULT_PATH:=''); (* URL zerlegen *)
		sep_char := CHR_TO_STRING(SEP);
		url_query := URL_DATA.QUERY;
		step_1 := 30;

		(* ---------------- Debug-Message -----------------------*)
		(*IF _debug_enable THEN
			LOG_CL.NEW_MSG := 'FILE_RRD1 - Start: DATE [~2]';
			LOG_CL.PRINTF[2] := DT_TO_STRING(DTI);
			LOG_MSG();
		END_IF;*)
		(* -----------------------------------------------------------------*)

	END_IF;

30:	(* LOG-Trigger verarbeiten *)
	trig_tmp := (TRIG_M AND NOT trig_m_last) OR trig_auto OR X.ADD_DATA_REQ;

	IF ENABLE = FALSE THEN (* ENABLE = 0 -> Log Stop *)
		X.ADD_COM := 00;
		step_1 := 00;

		(* ---------------- Debug-Message -----------------------*)
		(*IF _debug_enable THEN
			LOG_CL.NEW_MSG := 'FILE_RRD1 - Stop: DATE [~2]';
			LOG_CL.PRINTF[2] := DT_TO_STRING(DTI);
			LOG_MSG();
		END_IF;*)
		(* -----------------------------------------------------------------*)

	ELSIF ENABLE THEN
		IF trig_tmp OR trig_stored THEN (* manueller, automatischer oder externer Trigger *)
			trig_stored := FALSE;
			X.ADD_COM := 03; (* ADD DATA *)
			(* ---------------- Debug-Message -----------------------*)
			(*IF _debug_enable THEN
				LOG_CL.NEW_MSG := 'FILE_RRD1 - Trig: DATE [~2]';
				LOG_CL.PRINTF[2] := DT_TO_STRING(DTI);
				LOG_MSG();
			END_IF;*)
			(* -----------------------------------------------------------------*)
		ELSE
			X.ADD_COM := 04;	(* ADD DATA REQ *)
		END_IF;
	END_IF;

END_CASE;
X.ADD_DATA_REQ := FALSE; (* externe Anforderung rücksetzen *)

(* ##################################### *)

CASE step_2 OF

00:	IF X.UCB.BUF_COUNT >= USINT_TO_INT(X.ID_MAX) THEN (* genug Einträge vorhanden *)
		URL_DATA.QUERY := url_query; (* original Query wiederherstellen *)
		n := 1;
		WHILE n <= USINT_TO_INT(X.ID_MAX) DO
			X.UCB.D_MODE := 12; (* Element lesen und löschen *)
			UCB(DATA:=X.UCB);
			IF n < USINT_TO_INT(X.ID_MAX) THEN (* Trennzeichen hinzufügen *)
				X.UCB.D_STRING := CONCAT(X.UCB.D_STRING,sep_char);
			END_IF;
			IF LEN(X.UCB.D_STRING) + LEN(URL_DATA.QUERY) <= STRING_LENGTH THEN
				URL_DATA.QUERY := CONCAT(URL_DATA.QUERY,X.UCB.D_STRING); (* Query mit LOG-Daten ergänzen *)
				step_2 := 40;
			ELSE
				ERROR_T := BYTE#4; (* LOG-Daten können nicht in URL gepackt werden *)
				ERROR_C := DWORD#1;
				step_2 := 100;
			END_IF;
			n := n + 1;
		END_WHILE;;
	END_IF;

40:	IF DNS_CLIENT.DONE THEN
		step_2 := 60;
	ELSIF (DNS_CLIENT.ERROR > DWORD#0) THEN
		ERROR_C := DNS_CLIENT.ERROR; (* Fehlerbehandlung *)
		ERROR_T := BYTE#1;
		step_2 := 100;
	END_IF;

60:	IF HTTP_GET.DONE THEN
		n := UINT_TO_INT(HTTP_GET.BODY_START);
		IF R_BUF.BUFFER[n] <> BYTE#48 THEN (* ASCII '0' *)
			ERROR_C := DWORD#1;
			ERROR_T := BYTE#3;
		END_IF;
		step_2 := 100;

	ELSIF HTTP_GET.ERROR > DWORD#0 THEN (* Fehlerbehandlung *)
		ERROR_C := HTTP_GET.ERROR;
		ERROR_T := BYTE#2;
		step_2 := 100;
	END_IF;

100:	IF (NOT HTTP_GET.DONE) THEN (* UNLOCK HTTP DATA *)
		step_2 := SEL(ERROR_T = BYTE#0, 120,0);
	END_IF;

120:	IF NOT ENABLE THEN
		step_2 := 0;
	END_IF;

END_CASE;

HTTP_GET(IP_C:=IP_C,S_BUF:=S_BUF,R_BUF:=R_BUF,IP4:=DNS_CLIENT.IP4,GET:=step_2=60,MODE:=2,UNLOCK_BUF:=step_2=100,URL_DATA:=URL_DATA); (* HTTP_GET *)
DNS_CLIENT(IP_C:=IP_C, S_BUF:=S_BUF, R_BUF:=R_BUF, DOMAIN:=URL_DATA.DOMAIN, IP4_DNS:= DNS_IP4, ACTIVATE:=step_2=40); (* DNS-Client *)
IPC(IP:= 0, PORT:= 0 , TIME_OUT:= TIMEOUT, IP_C:= IP_C, S_BUF:= S_BUF, R_BUF:= R_BUF); (* IP_CONTROL *)

trig_m_last := TRIG_M;

(* revision history
ks	01. jan. 2011	rev 1.0
	original version

ks	13. may. 2011	rev 1.1
	ADD_DATA_REQ hinzugefügt

ks	26. july. 2011	rev 1.2
	code optimierung D_MODE 12 und bessere fehlerauswertung

ks	16. apr. 2012	rev 1.3
	neuer überarbeiteter Code
*)
END_FUNCTION_BLOCK

(* POU HTTP_GET, ST *)
FUNCTION_BLOCK HTTP_GET
VAR_IN_OUT
	URL_DATA : url;
	IP_C : IP_C; (* IP_Control Verwaltungsstruktur *)
	S_BUF : NETWORK_BUFFER;
	R_BUF : NETWORK_BUFFER;
END_VAR
VAR_INPUT
	IP4 : DWORD;
	GET : BOOL;
	MODE : BYTE := BYTE#2;
	UNLOCK_BUF : BOOL;
END_VAR
VAR_OUTPUT
	HTTP_STATUS : STRING;
	HEADER_START : UINT; (* HTTP Header (Message Header) *)
	HEADER_STOP : UINT; (* HTTP Header (Message Header) *)
	BODY_START : UINT; (* Message Body *)
	BODY_STOP : UINT; (* Message Body *)
	DONE : BOOL;
	ERROR : DWORD;
END_VAR
VAR
	READ_HTTP :	READ_HTTP;
	IP_FIFO : IP_FIFO;
	ip_state : BYTE;
	ip_id : BYTE;
	get_last : BOOL;
	ip4_stored : DWORD;
	state : INT;
	i : INT;
	http_1_1_host : BOOL;
	total_size : INT;
	text : STRING(STRING_LENGTH);
	delimiter2b : STRING(2);
	delimiter4b : STRING(4);
	del_end : STRING(4);
	del_pos : INT;
	idx : INT;
	rcv_timeout : BOOL;
	con_rdce : BOOL;

	(*LOG_MSG : LOG_MSG;
	_debug_enable : BOOL := TRUE;*)

END_VAR

(*

version 1.3	12. apr. 2011
programmer 	ks
tested by		ks

HTTP_GET führt eine HTTP Abfrage einer Web-Seite bei einem WEB_Server durch, und stellt die Daten ausbereitet zu verfügung
*)
CASE state OF
00:	IF GET AND NOT GET_LAST THEN (* auf positive Flanke SET warten *)
		state := 10;
		ip4_stored := IP4; (* aktuelle IP4 speichern *)
		DONE := FALSE;
		total_size := 0;
		HEADER_START := UINT#0;
		HEADER_STOP := UINT#0;
		BODY_START := UINT#0;
		BODY_STOP := UINT#0;
		HTTP_STATUS := '';
		ERROR := DWORD#0;
		ip_state := BYTE#1; (* Anmelden *)
		delimiter2b := '$0D$0A';
		delimiter4b := '$0D$0A$0D$0A';
	        	(*####################  DEBUG-MESSAGE  ###################################*)
		(*IF _debug_enable THEN
	       		LOG_CL.NEW_MSG := 'HTTP: S00 START /IP_ID ~4';
	            	LOG_CL.PRINTF[4]  := BYTE_TO_STRING(IP_ID);
	            	LOG_MSG();
	        	END_IF;*)
	        	(*########################################################################*)
	END_IF;

10:	IF ip_state = BYTE#3 THEN (* Bei IP_Control anmelden und auf freigabe warten *)
		idx := 0;
		text := CONCAT('GET ',URL_DATA.PATH);
		_STRING_TO_BUFFER(STR:=text,POS:=idx,PT:=ADR(S_BUF.BUFFER),SIZE:=SIZEOF(S_BUF.BUFFER)); (* GET path in buffer kopieren *)
		idx := idx + LEN(text);

		IF LEN(URL_DATA.QUERY) > 0 THEN
			S_BUF.BUFFER[idx] := 63; (* ASCII '?' *)
			idx := idx + 1;
			_STRING_TO_BUFFER(STR:=URL_DATA.QUERY,POS:=idx,PT:=ADR(S_BUF.BUFFER),SIZE:=SIZEOF(S_BUF.BUFFER)); (* QUERY in buffer kopieren *)
			idx := idx + LEN(URL_DATA.QUERY);
		END_IF;

		IF MODE >= BYTE#2 THEN (* gewünschte HTTP Version uebergeben *)
			text := ' HTTP/1.1';
		ELSE
			text := ' HTTP/1.0';
		END_IF;
		text := CONCAT(text,delimiter2b);
		_STRING_TO_BUFFER(STR:=text,POS:=idx,PT:=ADR(S_BUF.BUFFER),SIZE:=SIZEOF(S_BUF.BUFFER)); (* HTTP Version in buffer kopieren *)
		idx := idx + LEN(text);

		IF MODE = BYTE#1 THEN (* HTTP/1.0 mit persistenter Verbindung gewünscht *)
			text := CONCAT('Connection: Keep-Alive',delimiter2b); (* workaround für pcworx -> kein $0D$0A als Stringkonstante möglich *)
		ELSIF MODE = BYTE#3 THEN (* HTTP/1.1 ohne persistenter Verbindung gewünscht *)
			text := CONCAT('Connection: Close',delimiter2b); (* workaround für pcworx -> kein $0D$0A als Stringkonstante möglich *)
		ELSE
			text := '';
		END_IF;
		text := CONCAT(text,URL_DATA.HEADER);
		_STRING_TO_BUFFER(STR:=text,POS:=idx,PT:=ADR(S_BUF.BUFFER),SIZE:=SIZEOF(S_BUF.BUFFER)); (* HTTP Version in buffer kopieren *)
		idx := idx + LEN(text);

		text := CONCAT('Host: ',URL_DATA.DOMAIN);
		text := CONCAT(text,delimiter4b); (* workaround für pcworx -> kein $0D$0A als Stringkonstante möglich *)
		_STRING_TO_BUFFER(STR:=text,POS:=idx,PT:=ADR(S_BUF.BUFFER),SIZE:=SIZEOF(S_BUF.BUFFER)); (* HTTP Host in buffer kopieren *)
		idx := idx + LEN(text);

		(* IP Datenverkehr einrichten *)
		IF URL_DATA.PORT = WORD#0 THEN
			IP_C.C_PORT := WORD#80; (* Standard-Portnummer verwenden *)
		ELSE
			IP_C.C_PORT := URL_DATA.PORT; (* Portnummer aus URL verwenden *)
		END_IF;

		IP_C.C_IP := ip4_stored; (* IP eintragen *)
		IP_C.C_MODE := BYTE#0; (* Mode: TCP+AKTIV+PORT+IP *)
		IP_C.C_ENABLE := TRUE; (* Verbindungsaufbau freigeben *)
		IP_C.TIME_RESET := TRUE; (* Zeitueberwachung rücksetzen *)
		IP_C.R_OBSERVE := TRUE; (* Datenempfang ueberwachen *)
		S_BUF.SIZE := INT_TO_UINT(idx); (* Sendelänge eintragen *)
		R_BUF.SIZE := UINT#0; (* Empfangslänge rücksetzen *)

		state := 30;
	        	(*####################  DEBUG-MESSAGE  ###################################*)
	        	(*IF _debug_enable THEN
	        		LOG_CL.NEW_MSG := 'HTTP: S20 SEND /IP_ID ~4';
	            	LOG_CL.PRINTF[4]  := BYTE_TO_STRING(IP_ID);
	            	LOG_MSG();
	        	END_IF;*)
	        	(*########################################################################*)
	END_IF;

30:	rcv_timeout := (IP_C.ERROR AND DWORD#16#0000_FF00) = DWORD#16#0000_FF00;
	con_rdce :=     (IP_C.ERROR AND DWORD#16#FD00_0000) = DWORD#16#FD00_0000;

	IF S_BUF.SIZE = UINT#0 THEN
		IF total_size = 0 THEN
			IF R_BUF.SIZE > UINT#15 THEN; (* länge der empfangenen Daten prüfen *)

				(* HTTP HEADER Ende suchen -> durch $0D$A$0D$A erkennbar bei DEC RT-11,CP/M,MS-DOS,Windows *)
				del_end := '$0D$0A$0D$0A';
				del_pos := BUFFER_SEARCH(PT:=ADR(R_BUF.BUFFER),SIZE:=R_BUF.SIZE,STR:=del_end,POS:=0,IGN:=FALSE);

				(* kein Ende gefunden ? -> andere Ende-Codierung suchen *)
				IF del_pos = 0 THEN
					del_end := '$0A$0A';
					(* HTTP HEADER Ende suchen -> durch $0A$0A erkennbar bei Multics, Unix-Derivate,Mac OS X *)
					del_pos := BUFFER_SEARCH(PT:=ADR(R_BUF.BUFFER),SIZE:=R_BUF.SIZE,STR:=del_end,POS:=0,IGN:=FALSE);
				END_IF;

				IF del_pos > 0 THEN
					HEADER_START := UINT#0;
					HEADER_STOP := INT_TO_UINT(del_pos + LEN(del_end) - 1);
					TOTAL_SIZE := -1; (* HTTP Header empfangen aber noch keine gesamtlänge bekannt *)
				END_IF;
		                	(*####################  DEBUG-MESSAGE  ###################################*)
		                	(*IF _debug_enable THEN
		                   	LOG_CL.NEW_MSG := 'HTTP: S20 HEADER_START ~1 / HEADER_STOP ~2/IP_ID ~4';
		                   	LOG_CL.PRINTF[4]  := BYTE_TO_STRING(IP_ID);
		                   	LOG_CL.PRINTF[1]  := UINT_TO_STRING(HEADER_START);
		                   	LOG_CL.PRINTF[2]  := UINT_TO_STRING(HEADER_STOP);
		                   	LOG_MSG();
		                	END_IF;*)
		                	(*########################################################################*)

				(* HTTP Statuscode auswerten: (kann 1.0 oder 1.1 sein *)
				READ_HTTP(size:=HEADER_STOP,pos:=0,SRC:='',pt:=R_BUF.BUFFER);

				i := LEN(READ_HTTP.READ_HTTP);
				IF i > 7 THEN
					(* HTTP Version von HOST auswerten 1.0 oder 1.1 *)
					text:=MID(READ_HTTP.READ_HTTP,1,3);
					http_1_1_host := text = '1';

					(* Code und Meldung isolieren *)
					HTTP_STATUS := RIGHT(READ_HTTP.READ_HTTP,i-4);
				END_IF;

				(* positive HTTP Anfrage ? *)
				IF FIND(HTTP_STATUS,'200') > 0 THEN

					(* 'Content-Length: Wert einlesen auswerten *)
					READ_HTTP(size:=HEADER_STOP,pos:=0,SRC:='CONTENT-LENGTH',pt:=R_BUF.BUFFER);
					text:=READ_HTTP.READ_HTTP;

					IF LEN(text) >= 1 THEN
						IF IS_NUM(str:=text) THEN
							(* erwartete gesamtmenge an Bytes berechnen *)
							total_size := STRING_TO_INT(text) + UINT_TO_INT(HEADER_STOP) + 1;
                           					(*####################  DEBUG-MESSAGE  ###################################*)
                           					(*IF _debug_enable THEN
                              					LOG_CL.NEW_MSG := 'HTTP: S20 HEADER ~1, BODY ~2 TOTAL ~3 /IP_ID ~4';
                             					LOG_CL.PRINTF[4]  := BYTE_TO_STRING(IP_ID);
                               					LOG_CL.PRINTF[1]  := UINT_TO_STRING(HEADER_STOP);
                               					LOG_CL.PRINTF[2]  := INT_TO_STRING(TOTAL_SIZE-UINT_TO_INT(HEADER_STOP));
                               					LOG_CL.PRINTF[3]  := INT_TO_STRING(TOTAL_SIZE);
                              					LOG_MSG();
                          					END_IF;*)
                          					(*########################################################################*)
						END_IF;
					END_IF;
				ELSE
					ERROR := DWORD#16#000000FC; (* Fehler durch HTTP-Statuscodes *)
				END_IF;
			END_IF;
		(* 1. bei bekannter Content-Length wird nach erhalt der erwartenen Daten die verbindung beendet *)
		(* 2. bei persistenter Verbindung muss bei unbekannter Datenmenge auf Receive-Timeout gewartet werden *)
		(* 3. wenn nach datenempfang die verbindung vom host unterbrochen wird *)
		ELSIF (R_BUF.SIZE >= INT_TO_UINT(total_size)) OR
			(R_BUF.SIZE > UINT#0 AND total_size < 0 AND ((rcv_timeout OR con_rdce) OR (IP_C.C_STATE = BYTE#1))) THEN

			IF R_BUF.SIZE - 1 > HEADER_STOP THEN (* BODY Daten vorhanden *)
				BODY_START := HEADER_STOP + UINT#1;
				BODY_STOP := R_BUF.SIZE - 1;
		                	(*####################  DEBUG-MESSAGE  ###################################*)
		                	(*IF _debug_enable THEN
		                   	LOG_CL.NEW_MSG := 'HTTP: S20 BODY ~1, START ~2 END ~3 /IP_ID ~4';
		                   	LOG_CL.PRINTF[4]  := BYTE_TO_STRING(IP_ID);
		                   	LOG_CL.PRINTF[1]  := UINT_TO_STRING(HEADER_STOP);
		                   	LOG_CL.PRINTF[2]  := UINT_TO_STRING(BODY_START);
		                   	LOG_CL.PRINTF[3]  := UINT_TO_STRING(BODY_STOP);
		                   	LOG_MSG();
		               	END_IF;*)
		               	(*########################################################################*)
			END_IF;

			DONE := TRUE;
			IP_C.C_ENABLE := FALSE; (* Verbindung abbauen *)
			state := 40;
            		(*####################  DEBUG-MESSAGE  ###################################*)
            		(*IF _debug_enable THEN
                			LOG_CL.NEW_MSG := 'HTTP: S30 OK /IP_ID ~4';
                			LOG_CL.PRINTF[4]  := BYTE_TO_STRING(IP_ID);
                			LOG_MSG();
            		END_IF;*)
            		(*########################################################################*)
		END_IF;
	END_IF;

	IF IP_C.ERROR <> DWORD#0 THEN
		(* bei unbekannter Content-size ist nicht bekannt ob bzw wieviele Telegramme noch folgen werden *)
		(* darum wird nach receive-timeout oder Remote disconnect error der fehler wieder ausgefiltert (logischer fehler) *)
		IF rcv_timeout AND DONE THEN
			IP_C.ERROR := IP_C.ERROR AND DWORD#16#FFFF_00FF; (* Fehler wieder rücksetzen *)
		ELSIF con_rdce AND DONE THEN
			IP_C.ERROR := IP_C.ERROR AND DWORD#16#00FF_FFFF; (* Fehler wieder rücksetzen *)
		ELSE
			ERROR := IP_C.ERROR;
		END_IF;
	END_IF;

	IF ERROR > DWORD#0 THEN
		IP_C.C_ENABLE := FALSE; (* Verbindungsaufbau sperren *)
		state := 40;
	        	(*####################  DEBUG-MESSAGE  ###################################*)
	        	(*IF _debug_enable THEN
	            	LOG_CL.NEW_MSG := 'HTTP: S30 ERROR ~1 /IP_ID ~4';
	            	LOG_CL.PRINTF[1]  := DWORD_TO_STRING(ERROR);
	            	LOG_CL.PRINTF[4]  := BYTE_TO_STRING(IP_ID);
	            	LOG_MSG();
	        	END_IF;*)
	        	(*########################################################################*)
	END_IF;

40:	IF (UNLOCK_BUF OR NOT DONE) THEN (* Warten auf Release und Verbindung beendet -> IP_ID vom Stack nehmen *)
		IP_STATE := BYTE#4; (* Abmelden *)
		DONE := FALSE;
		state := 0;
	END_IF;
END_CASE;

get_last := GET; (* letzten Status sichern zur Flankenerkennung *)

IP_FIFO(FIFO:=IP_C.FIFO,STATE:=ip_state,ID:=ip_id); (* IP_FIFO *)

(* revision history
ks	18. oct. 2008	rev 1.0
	original version

ks	20. oct. 2009	rev 1.1
	Fehler bei body-suche bei $0a$0a korrigiert,Codeoptimierung,
	new VAR del_pos , del_end (Networkbuffer und Buffer-funktionen auf Basis 0)

ks	28. oct. 2009	rev 1.2
	über url.header können zusätzliche header-infos übergeben werden

ks	12. apr. 2011	rev 1.3
	verbesserte fehlererkennung und fehlerkorrektur bei buffer_to_string
*)
END_FUNCTION_BLOCK

(* POU READ_HTTP, ST *)
FUNCTION_BLOCK READ_HTTP
VAR_INPUT
	SIZE : UINT;
	POS : INT;
	SRC : STRING;
END_VAR
VAR_IN_OUT
	PT : NW_BUF_LONG;
END_VAR
VAR_OUTPUT
	READ_HTTP : STRING(STRING_LENGTH);
END_VAR
VAR
	index : INT;
	s1 : INT;
	e1 : INT;
	stop : INT;
END_VAR

(*

version 1.1 20. oct. 2009
programmer 	ks
tested by	ks

READ_HTTP wertet die Informationen einer HTTP-Request aus, und stellt die Daten zu Verfügung.
*)
stop := UINT_TO_INT(SIZE) - 1;

IF LEN(SRC) = 0 THEN
	(* wenn kein Suchbegriff vorhanden ist, dann den HTTP-STATUS auswerten *)
	SRC := 'HTTP/'; (* neuer Suchbegriff *)
ELSE
	(* gesuchten Parametertext ergänzen *)
	SRC := CONCAT(SRC,': ');
END_IF;

s1 := BUFFER_SEARCH(pt:=ADR(PT),SIZE:=SIZE,STR:=SRC,POS:=POS,IGN:=TRUE);

IF s1 >= 0 THEN (* Text found *)
	e1 := s1;

	(* search start of line *)
	index := s1 - 1;
	WHILE (index > 0) DO
		IF pt[index] < BYTE#32 THEN EXIT; END_IF;
		s1 := s1 - 1;
		index := index - 1;
	END_WHILE;

	(* search end of line *)
	index := e1 + 1;
	WHILE (index <= stop) DO
		IF pt[index] < BYTE#32 THEN EXIT; END_IF;
		e1 := e1 + 1;
		index := index + 1;
	END_WHILE;

	s1 := s1 + LEN(SRC); (* 'suchbegriff: ' nicht mitkopieren *)

	(* copy string *)
	READ_HTTP := BUFFER_TO_STRING(PT:=ADR(PT),SIZE:=SIZE,START:=s1,STOP:=e1);
ELSE
	READ_HTTP := '';
END_IF;

(* revision history

ks	18. oct. 2008	rev 1.0
	original version

ks	20. oct. 2009	rev 1.1
	Networkbuffer und Buffer-funktionen auf Basis 0

*)
END_FUNCTION_BLOCK

(* POU DNS_DYN_DEMO, CFC *)
PROGRAM DNS_DYN_DEMO
VAR
	DNS_DYN : DNS_DYN;
	IP_C : IP_C;
	S_BUF : NETWORK_BUFFER;
	R_BUF : NETWORK_BUFFER;
	IP_CONTROL : IP_CONTROL;
	enable: BOOL;
	done : BOOL;
	error_c : DWORD;
	error_t : BYTE;
	busy : BOOL;
	COUNT_DR: COUNT_DR;
	z: DWORD;

	GET_WAN_IP : GET_WAN_IP;
	t1: TON;
	done2 : BOOL;
	error_c2 : DWORD;
	error_t2 : BYTE;
	update : BOOL;
	new_ip: BOOL;
	wan_ip4: DWORD;
END_VAR
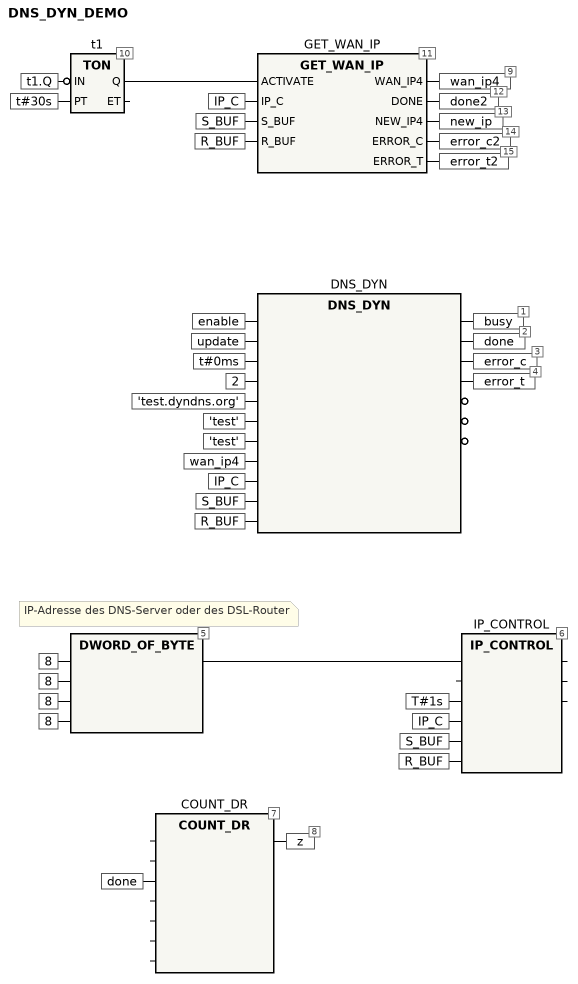
_CFC_ (* Continuous Function Chart, elements in execution order *)
#0 DNS_DYN:DNS_DYN(enable, update, t#0ms, 2, 'test.dyndns.org', 'test', 'test', wan_ip4, IP_C, S_BUF, R_BUF)
#1 busy <= #0.out 1
#2 done <= #0.out 2
#3 error_c <= #0.out 3
#4 error_t <= #0.out 4
#5 DWORD_OF_BYTE(8, 8, 8, 8)
#6 IP_CONTROL:IP_CONTROL(#5, -, T#1s, IP_C, S_BUF, R_BUF)
#7 COUNT_DR:COUNT_DR(-, -, done, -, -, -, -)
#8 z <= #7
#9 wan_ip4 <= #11.WAN_IP4
#10 t1:TON(IN: NOT t1.Q, PT: t#30s)
#11 GET_WAN_IP:GET_WAN_IP(ACTIVATE: #10.Q, IP_C: IP_C, S_BUF: S_BUF, R_BUF: R_BUF)
#12 done2 <= #11.DONE
#13 new_ip <= #11.NEW_IP4
#14 error_c2 <= #11.ERROR_C
#15 error_t2 <= #11.ERROR_T
(* IP-Adresse des DNS-Server oder des DSL-Router *)
_END_CFC_
END_PROGRAM

(* POU DNS_DYN, ST *)
FUNCTION_BLOCK DNS_DYN
VAR_IN_OUT
	IP_C : IP_C; (* IP_Control Verwaltungsstruktur *)
	S_BUF : NETWORK_BUFFER;
	R_BUF : NETWORK_BUFFER;
END_VAR
VAR_INPUT
	ENABLE : BOOL;
	UPDATE : BOOL;
	T_UPDATE : TIME := T#1h;
	MODE : BYTE;
	HOSTNAME : STRING(30);
	USERNAME : STRING(20);
	PASSWORD : STRING(20);
	IP4 : DWORD;
END_VAR
VAR_OUTPUT
	BUSY : BOOL;
	DONE : BOOL;
	ERROR_C : DWORD;
	ERROR_T : BYTE;
END_VAR
VAR
	DNS_CLIENT : DNS_CLIENT;
	HTTP_GET : HTTP_GET;
	BASE64_ENCODE_STR : BASE64_ENCODE_STR;
	URL_DATA : url;
	update_last : BOOL;
	state : INT;
	base64_done : BOOL;
	s1 : STRING(144);
	s2 : STRING(192);
	w : TON;
END_VAR

(*

version 1.2		02. dec. 2009
programmer 		ks
tested by		ks

YAHOO_WEATHER lädt vom Yahoo-Webserver einen Wetter RSS-Feed und analysiert die Daten und legt diese in einem Array ab
*)
CASE state OF

00:	IF ENABLE AND ((UPDATE AND NOT update_last) OR w.Q) THEN
		state := 20;
		DONE := FALSE;
		BUSY := TRUE;
		ERROR_C := DWORD#0;
		ERROR_T := BYTE#0;

		IF MODE = 0 THEN (* dyndns.org *)
			s2 := CONCAT('http://members.dyndns.org/nic/update?hostname=',HOSTNAME);
		ELSE (* selfhost.de *)
			s2 := 'http://carol.selfhost.de/nic/update?hostname=1';
		END_IF;
		IF IP4 > 0 THEN (* parametrierte IP verwenden *)
			s1 := CONCAT('&myip=',IP4_TO_STRING(IP4));
			s2 := CONCAT(s2,s1);
		END_IF;
		URL_DATA:=STRING_TO_URL(STR:=s2, DEFAULT_PROTOCOL:='', DEFAULT_PATH:=''); (* URL for DNS UND HTTP-GET *)
		s1 := CONCAT(USERNAME,':');
		s1 := CONCAT(s1,PASSWORD); (* BASE64 Encode Text *)
	END_IF;

20:	IF DNS_CLIENT.DONE THEN (* DNS_CLIENT *)
			state := 40;
	ELSIF (DNS_CLIENT.ERROR > DWORD#00) THEN (* Fehlerbehandlung *)
		ERROR_C := DNS_CLIENT.ERROR;
		ERROR_T := BYTE#01;
		BUSY := FALSE;
		state := 0;
	END_IF;

40: IF base64_done THEN (* BASE64 Encode beendet ? *)
		s1 := CONCAT('Authorization: Basic ',s2);
		s1 := CONCAT(s1,'$0D$0AUser-Agent: x$0D$0A');
		URL_DATA.HEADER := s1;
		state := 60;
	END_IF;

60:	IF HTTP_GET.DONE THEN
		state := 0;
		BUSY := FALSE;
		DONE := TRUE;

		(* !! Codes !!
		Successful Updates: 		good , nchg
		Update Syntax Errors:		badsys , badagent
		Account-Related Errors:		badauth , !donator
		Hostname-Related Errors:	notfqdn , nohost , !yours , numhost , abuse
		Server Error Conditions:	dnserr , 911
		*)
		s2 := BUFFER_TO_STRING(PT:=ADR(R_BUF.BUFFER),SIZE:=SIZEOF(R_BUF.BUFFER),START:=HTTP_GET.BODY_START + 3,STOP:=HTTP_GET.BODY_STOP - 7);
		IF FIND(s2,'good') = 0 THEN
			IF FIND(s2,'nochg') = 0 THEN
				ERROR_C := DWORD#1;
				ERROR_T := BYTE#03;
				DONE := FALSE;
			END_IF;
		END_IF;
	ELSIF (HTTP_GET.ERROR > DWORD#00) THEN (* Fehlerbehandlung *)
		ERROR_C := HTTP_GET.ERROR;
		ERROR_T := BYTE#02;
		BUSY := FALSE;
		state := 0;
	END_IF;

END_CASE;

DNS_CLIENT(IP_C:=IP_C,	S_BUF:=S_BUF, R_BUF:=R_BUF,DOMAIN:=URL_DATA.DOMAIN, IP4_DNS:=0, ACTIVATE:=state=20); (* DNS_CLIENT *)
HTTP_GET( IP_C:=IP_C, S_BUF:=S_BUF, R_BUF:=R_BUF, IP4:=DNS_CLIENT.IP4, GET:=state=60, MODE:=2, UNLOCK_BUF:=state<>60,URL_DATA:=URL_DATA); (* HTTP_GET *)
BASE64_ENCODE_STR( RUN:=state=40, STR1:=s1, STR2:=s2, DONE=>base64_done); (* BASE64 Encode *)

IF T_UPDATE > T#0ms THEN w(IN:=state=0, PT:=T_UPDATE); END_IF;
update_last := UPDATE;

(* revision history
ks	01. jan. 2010	rev 1.0
	original version

*)
END_FUNCTION_BLOCK

(* POU GET_WAN_IP, ST *)
FUNCTION_BLOCK GET_WAN_IP
VAR_IN_OUT
	IP_C : IP_C; (* IP_Control Verwaltungsstruktur *)
	S_BUF : NETWORK_BUFFER;
	R_BUF : NETWORK_BUFFER;
END_VAR
VAR_INPUT
	ACTIVATE : BOOL;
END_VAR
VAR_OUTPUT
	WAN_IP4 : DWORD;
	DONE : BOOL;
	NEW_IP4 : BOOL;
	ERROR_C : DWORD;
	ERROR_T : BYTE;
END_VAR
VAR
	URL_DATA : url;
	DNS_CLIENT : DNS_CLIENT;
	HTTP_GET : HTTP_GET;
	activate_last : BOOL;
	wan_ip4_last : DWORD;
	state : INT;
	st_ip : STRING(120);
	i1 :	INT;
	p1 : INT;
	p2 : INT;
	p3 : INT;
END_VAR

(*
version 1.1	28. dec. 2009
programmer 	ks
tested by	ks

GET_WAN_IP ermittelt die aktuelle WAN-IP (Internet-Adresse)
*)
CASE state OF

00:
	IF ACTIVATE AND NOT activate_last THEN
		state := 20;
		DONE := FALSE;
		ERROR_C := DWORD#0;
		ERROR_T := BYTE#0;
	END_IF;

20: (* URL for DNS UND HTTP-GET *)
	URL_DATA := STRING_TO_URL(STR:='checkip.dyndns.com',DEFAULT_PROTOCOL:='',DEFAULT_PATH:='');
	state := 40;

40:
	IF DNS_CLIENT.DONE THEN
		state := 60;
	ELSIF (DNS_CLIENT.ERROR > DWORD#00) THEN
		(* Fehlerbehandlung *)
		ERROR_C := DNS_CLIENT.ERROR;
		ERROR_T := BYTE#01;
		state := 100;
	END_IF;

60:
	IF HTTP_GET.DONE THEN
		state := 80;
	ELSIF (HTTP_GET.ERROR > DWORD#00) THEN
		(* Fehlerbehandlung *)
		ERROR_C := HTTP_GET.ERROR;
		ERROR_T := BYTE#02;
		state := 100;
	END_IF;

80:
	(* Als Antwort wird folgende HTML Seite empfangen , hier muss die IP-Adresse herauskopiert werden *)
	(* <html><head><title>Current IP Check</title></head><body>Current IP Address: 85.127.217.33</body></html> *)
	st_ip := '';
	p1 := 0;
	FOR i1 := UINT_TO_INT(HTTP_GET.BODY_START) TO UINT_TO_INT(HTTP_GET.BODY_STOP) DO
		IF R_BUF.BUFFER[i1] = BYTE#58 THEN (* suche ':' *)
			p1 := i1 + 2;
			EXIT;
		END_IF;
	END_FOR;

	p3 := p1 + 15;
	IF p1 > 0 AND p3 < UINT_TO_INT(HTTP_GET.BODY_STOP) THEN
		FOR p2 := p1 TO p3 DO
			IF R_BUF.BUFFER[p2] <> BYTE#60 THEN (* suche '<' *)
				st_ip := CONCAT(st_ip,CHR_TO_STRING(C:=R_BUF.BUFFER[p2]));
			ELSE
				EXIT;
			END_IF;
		END_FOR;
	END_IF;

	WAN_IP4 := IP4_DECODE(STR:=st_ip);

	IF WAN_IP4 <> DWORD#0 THEN
		DONE := TRUE;
		NEW_IP4 := WAN_IP4 <> wan_ip4_last;
		wan_ip4_last := WAN_IP4;
	ELSE
		ERROR_C := DWORD#01; (* keine gültige IP gefunden *)
		ERROR_T := BYTE#03;
	END_IF;
	state := 100;

100:
	(* UNLOCK HTTP DATA *)
	IF (NOT HTTP_GET.DONE) THEN
		state := 0;
		DONE := ERROR_T = BYTE#0;
	END_IF;

END_CASE;

(* ---------------- DNS --------------- *)
DNS_CLIENT(	IP_C:=IP_C,
			S_BUF:=S_BUF,
			R_BUF:=R_BUF,
			DOMAIN:=URL_DATA.DOMAIN,
			IP4_DNS:=DWORD#00,
			ACTIVATE:=state=40 (* DNS Start *)
			);
(* nicht oder nicht direkt verwendete Parameter *)
(* DWORD :=DNS_CLIENT.IP4;
   BOOL  :=DNS_CLIENT.DONE;
   BYTE  :=DNS_CLIENT.ERROR; *)
(* -------------------------------------*)

(* ------------- HTTP_GET --------------- *)

HTTP_GET(	IP_C:=IP_C,
			S_BUF:=S_BUF,
			R_BUF:=R_BUF,
			IP4:=DNS_CLIENT.IP4,
			GET:=state=60,
			MODE:=BYTE#2, (* HTTP 1.1 mit persistenter Verbindung *)
			UNLOCK_BUF:=state=100,
			URL_DATA:=URL_DATA
			);

(* nicht oder nicht direkt verwendete Parameter *)
(*STRING := HTTP_GET.HTTP_STATUS;
  UINT :=HTTP_GET.HEADER_START;
  UINT :=HTTP_GET.HEADER_STOP;
  UINT :=HTTP_GET.BODY_START;
  UINT :=HTTP_GET.BODY_STOP;
  BOOL :=HTTP_GET.DONE;
  BYTE :=HTTP_GET.ERROR;
*)
(* -------------------------------------*)

activate_last := ACTIVATE;

(* revision history
ks	28. dec 2009	rev 1.1
	original version

*)
END_FUNCTION_BLOCK

(* POU DNS_REV_DEMO, CFC *)
PROGRAM DNS_REV_DEMO
VAR
	DNS_REV_CLIENT: DNS_REV_CLIENT;
	IP_C : IP_C;
	S_BUF : NETWORK_BUFFER;
	R_BUF : NETWORK_BUFFER;
	IP_CONTROL : IP_CONTROL;
	activate : BOOL := TRUE;
	done : BOOL;
	error: DWORD;
	domain: STRING;
END_VAR
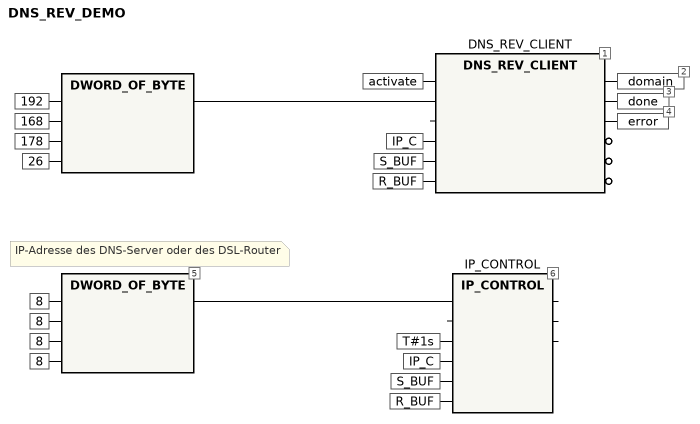
_CFC_ (* Continuous Function Chart, elements in execution order *)
#0 DWORD_OF_BYTE(192, 168, 178, 26)
#1 DNS_REV_CLIENT:DNS_REV_CLIENT(activate, #0, -, IP_C, S_BUF, R_BUF)
#2 domain <= #1.out 1
#3 done <= #1.out 2
#4 error <= #1.out 3
#5 DWORD_OF_BYTE(8, 8, 8, 8)
#6 IP_CONTROL:IP_CONTROL(#5, -, T#1s, IP_C, S_BUF, R_BUF)
(* IP-Adresse des DNS-Server oder des DSL-Router *)
_END_CFC_
END_PROGRAM

(* POU DNS_REV_CLIENT, ST *)
FUNCTION_BLOCK DNS_REV_CLIENT
VAR_IN_OUT
	IP_C : IP_C; (* IP_Control Verwaltungsstruktur *)
	S_BUF : NETWORK_BUFFER;
	R_BUF : NETWORK_BUFFER;
END_VAR
VAR_INPUT
	ACTIVATE : BOOL;
	IP4 : DWORD;
	IP4_DNS : DWORD;
END_VAR
VAR_OUTPUT
	DOMAIN : STRING;
	DONE : BOOL;
	ERROR : DWORD;
END_VAR
VAR
	IP_FIFO : IP_FIFO;
	ip_state : BYTE;
	ip_id : BYTE;
	state : INT;
	ip4_copy : DWORD;
	d : STRING(27);
	activate_last : BOOL;
	i : INT;
	dl : INT;
	p1 : INT;
	char : BYTE;
	char_count : INT;
	tid : BYTE;
END_VAR

(*
version 1.0	28. dec. 2009
programmer 	ks
tested BY	ks

DNS_REV_CLIENT führt eine Reverse-Domain-Name Abfrage durch, und ermittelt aus einer IP-Adresse den zugehörigen Domain-Namen.

*)
(* Domain Name System (query) *)

CASE state OF
00: (* auf positive Flanke GET warten *)
	IF ACTIVATE AND NOT activate_last THEN
		ERROR := DWORD#0;
		ip4_copy := ip4; (* IP4 sichern *)
		ip_state := BYTE#1;
		DOMAIN := '';
		DONE := FALSE;

		d := '';
		FOR i := 1 TO 4 DO
			d := CONCAT(d,BYTE_TO_STRING(DWORD_TO_BYTE(IP4)));
			d := CONCAT(d,'.');
			IP4 := ROR(IP4,8);
		END_FOR;
		d := CONCAT(d,'in-addr.arpa');
		state := 10;
	END_IF;

10: (* Bei IP_Control anmelden *)
	IF ip_state = BYTE#3 THEN
		dl := LEN(d);

		(* sendebuffer initialisieren *)
		char_count := 17 + dl;
		FOR i := 0 TO char_count DO
			S_BUF.BUFFER[i] := BYTE#00;
		END_FOR;

		tid := UINT_TO_BYTE(BYTE_TO_UINT(tid) + UINT#1);
		S_BUF.BUFFER[01] := tid; (* Transaction ID lowbyte *)
		S_BUF.BUFFER[02] := BYTE#16#01; (* Flags: highbyte *)
		S_BUF.BUFFER[05] := BYTE#16#01; (* Questions: lowbyte *)

		(* den servernamen von hinten nach vorne bearbeiten *)
		i := dl + 12;
		char_count := 0;

		WHILE i > 12 DO
			char := CODE(STR:=d,POS:=i - 12);

			(* prüfe auf haupt/sub domänen namens-teiler "." *)
			IF char = BYTE#46 THEN
				(* anstelle des teilers "." wird die länge des erkannten haupt/sub domänennames eingetragen *)
				S_BUF.BUFFER[i] := INT_TO_BYTE(char_count);
				char_count := 0;
			ELSE
				S_BUF.BUFFER[i] := char; (* char in buffer eintragen *)
				char_count := char_count + 1; (* anzahl char zählen *)
			END_IF;
			i := i - 1;
		END_WHILE;

		S_BUF.BUFFER[i] := INT_TO_BYTE(char_count); (* längenangabe des ganz linken (ersten) domänennamens eintragen *)
		i := dl + 15; (* position hinter dem servernamen *)
		S_BUF.BUFFER[i] := BYTE#12; (* Type: PTR (Domain name pointer) lowbyte *)
		i := i + 2;
		S_BUF.BUFFER[i] := BYTE#01; (* Class: IN lowbyte *)
		i := i + 1;

		(* IP Datenverkehr einrichten *)
		IP_C.C_PORT := WORD#53; (* Portnummer eintragen *)
		IP_C.C_IP := IP4_DNS; (* IP eintragen *)
		IP_C.C_MODE := BYTE#1; (* Mode: UDP+AKTIV+PORT+IP *)
		IP_C.C_ENABLE := TRUE; (* Verbindungsaufbau freigeben *)
		IP_C.TIME_RESET := TRUE; (* Zeitueberwachung rücksetzen *)
		IP_C.R_OBSERVE  := TRUE; (* Datenempfang ueberwachen *)
		S_BUF.SIZE := INT_TO_UINT(i); (* sendelänge eintragen *)
		R_BUF.SIZE := UINT#0; (* Empfangslänge rücksetzen *)
		state := 30;
	END_IF;

30:
	IF IP_C.ERROR <> DWORD#00 THEN
		ERROR := IP_C.ERROR;
	(* prüfe ob antwort telegramm die richtige Transaction-ID und mindestlänge hat *)
	ELSIF (S_BUF.SIZE = UINT#0) AND (tid = R_BUF.BUFFER[1]) AND (R_BUF.SIZE >= INT_TO_UINT(i+12)) THEN

		(* prüfe Return code der Flags. 4 bits *)
		ERROR := BYTE_TO_DWORD(R_BUF.BUFFER[3] AND BYTE#2#0000_1111);

		IF ERROR = DWORD#00 THEN

			i := R_BUF.SIZE - 2;
			WHILE R_BUF.BUFFER[i] > 0 DO
				IF i = 0 THEN EXIT; END_IF;
				i := i - 1;
			END_WHILE;

			i := i + 2;
			p1 := i + 1;
			WHILE i < R_BUF.SIZE DO
				dl := R_BUF.BUFFER[i];
				IF dl > 0 THEN
					R_BUF.BUFFER[i] := BYTE#46;
					i := i + dl + 1;
				ELSE
					DOMAIN := BUFFER_TO_STRING(PT:=ADR(R_BUF.BUFFER),SIZE:=SIZEOF(R_BUF.BUFFER),START:=p1,STOP:=i-1);
					EXIT;
				END_IF;
			END_WHILE;
			state := 0;
			DONE := TRUE;
		END_IF;
	END_IF;

	IF ERROR <> DWORD#0 THEN
		state := 0;
	END_IF;

	IF state = 0 THEN
		IP_C.R_OBSERVE := FALSE; (* Datenempfang ueberwachen *)
		ip_state := BYTE#4; (* Abmelden *)
	END_IF;

END_CASE;

activate_last := ACTIVATE; (* letzten Status sichern zur Flankenerkennung *)

(* IP_FIFO *)
IP_FIFO(FIFO:=IP_C.FIFO,STATE:=ip_state,ID:=ip_id);

(* revision history

ks	28. dec. 2009	rev 1.0
	original version

*)


(*----------------------------------------------------------------------------------------------------------------*)
(* Flags: 0x0100 (Standard query)                                                                                            *)
(* 0... .... .... .... = Response: Message is a query                                                                   *)
(* .000 0... ....  = Opcode: Standard query (0)                                                                          *)
(* .... ..0. .... .... = Truncated: Message is not truncated                                                          *)
(* .... ...1 .... .... = Recursion desired: Do query recursively                                                    *)
(* .... .... .0.. .... = Z: reserved (0)                                                                                                  *)
(* .... .... ...0 .... = Non-authenticated data OK: Non-authenticated data is unacceptable *)
(*-----------------------------------------------------------------------------------------------------------------*)

(*
Errorcodes  Description	References 
000	No error. 		 	The request completed successfully.
001	Format error. 		The name server was unable to interpret the query. 
002	Server failure.  	The name server was unable to process this query due to a problem with the name server. 
003	Name Error. 	 	Meaningful only for responses from an authoritative name server, this code signifies that the domain name referenced in the query does not exist.
004	Not Implemented. 	The name server does not support the requested kind of query.
005	Refused. 			The name server refuses to perform the specified operation for policy reasons.
  						 For example, a name server may not wish to provide the information to the particular requester, or a name server may not wish to perform a particular operation (e.g., zone transfer) for particular data.
006	YXDomain.			Name Exists when it should not. 
007	YXRRSet. RR			Set Exists when it should not. 
008	NXRRSet. RR			Set that should exist does not. 
009	NotAuth.			Server Not Authoritative for zone. 
010	NotZone,			Name not contained in zone. 
255	Timeout				No Response  
*)   
END_FUNCTION_BLOCK

(* POU DNS_SNTP_SYSLOG_DEMO, CFC *)
PROGRAM DNS_SNTP_SYSLOG_DEMO
VAR
	IP_C : IP_C;
	S_BUF : NETWORK_BUFFER;
	R_BUF : NETWORK_BUFFER;
	IP_CONTROL_1: IP_CONTROL;
	DNS_CLIENT : DNS_CLIENT;
	SNTP_CLIENT: SNTP_CLIENT;
	SNTP_SERVER: SNTP_SERVER;
	COUNT_DR: COUNT_DR;
	RTC_2: RTC_2;
	count_cycles: DWORD;
	dns_error: DWORD;
	sntp_error: DWORD;
	freigabe: BOOL;
	dso: BOOL;
	xms: INT;
	sntp_srv_enable: BOOL;
	cur_UDT: DT;
	cur_LDT: DT;
	SYS_LOG: SYS_LOG;
	sys_log_option: BYTE := 2#0000_0100;
	TON_1: TON;
	tp_sys_log: BOOL;
	error_sys_log: DWORD;
	sys_time: TIME;
END_VAR
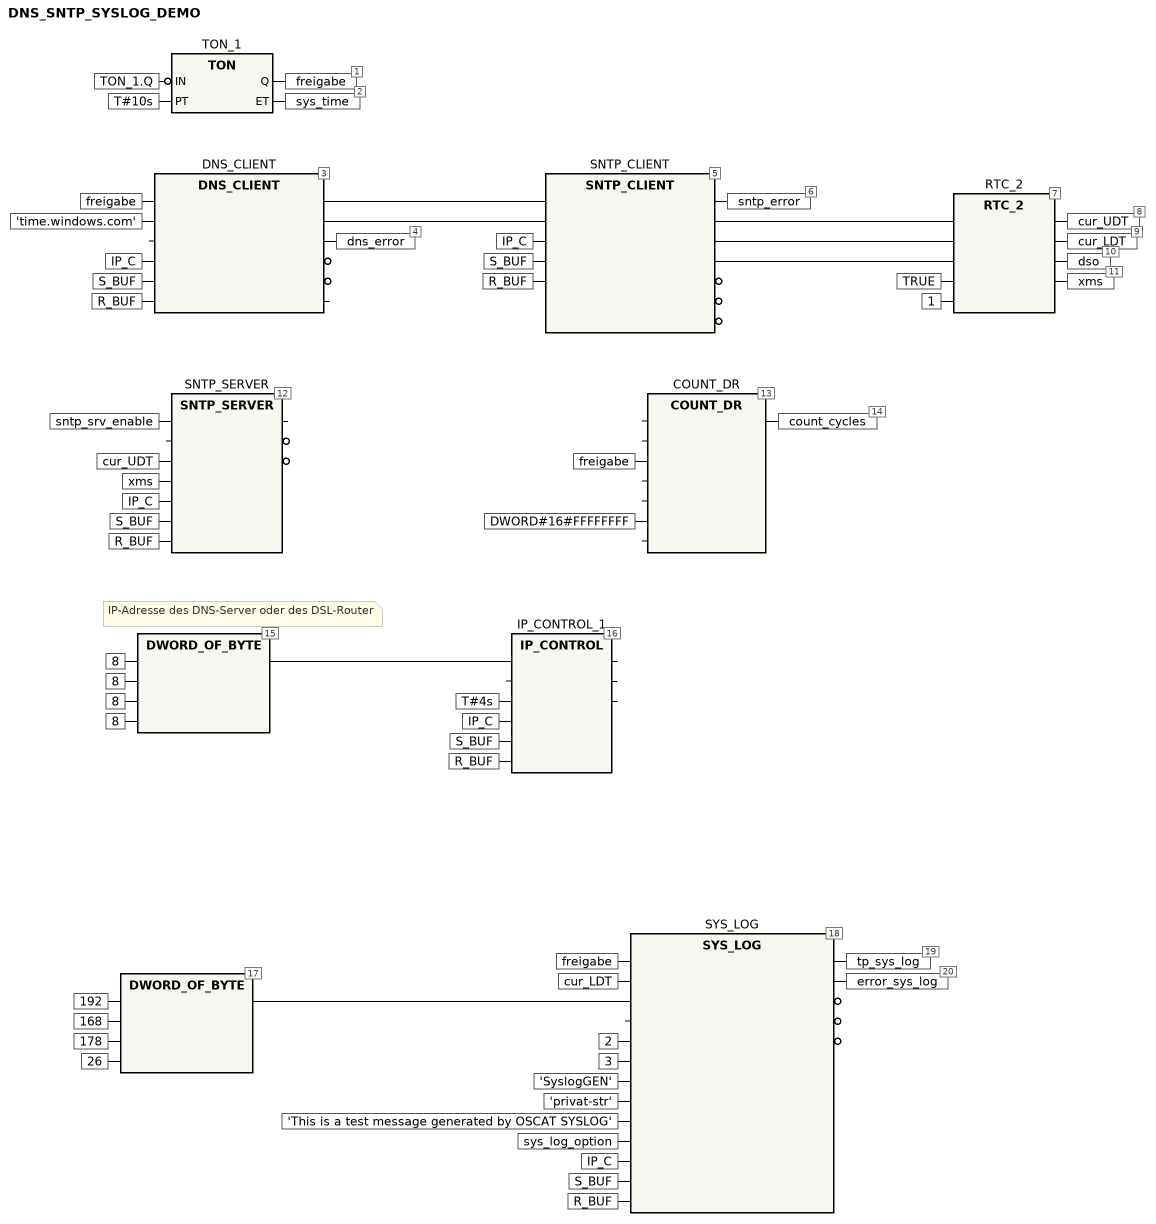
_CFC_ (* Continuous Function Chart, elements in execution order *)
#0 TON_1:TON(IN: NOT TON_1.Q, PT: T#10s)
#1 freigabe <= #0.Q
#2 sys_time <= #0.ET
#3 DNS_CLIENT:DNS_CLIENT(freigabe, 'time.windows.com', -, IP_C, S_BUF, R_BUF)
#4 dns_error <= #3.out 3
#5 SNTP_CLIENT:SNTP_CLIENT(#3.out 1, #3.out 2, IP_C, S_BUF, R_BUF)
#6 sntp_error <= #5.out 1
#7 RTC_2:RTC_2(#5.out 2, #5.out 3, #5.out 4, TRUE, 1)
#8 cur_UDT <= #7.out 1
#9 cur_LDT <= #7.out 2
#10 dso <= #7.out 3
#11 xms <= #7.out 4
#12 SNTP_SERVER:SNTP_SERVER(sntp_srv_enable, -, cur_UDT, xms, IP_C, S_BUF, R_BUF)
#13 COUNT_DR:COUNT_DR(-, -, freigabe, -, -, DWORD#16#FFFFFFFF, -)
#14 count_cycles <= #13
#15 DWORD_OF_BYTE(8, 8, 8, 8)
#16 IP_CONTROL_1:IP_CONTROL(#15, -, T#4s, IP_C, S_BUF, R_BUF)
#17 DWORD_OF_BYTE(192, 168, 178, 26)
#18 SYS_LOG:SYS_LOG(freigabe, cur_LDT, #17, -, 2, 3, 'SyslogGEN', 'privat-str', 'This is a test message generated by OSCAT SYSLOG', sys_log_option, IP_C, S_BUF, R_BUF)
#19 tp_sys_log <= #18.out 1
#20 error_sys_log <= #18.out 2
(* IP-Adresse des DNS-Server oder des DSL-Router *)
_END_CFC_
END_PROGRAM

(* POU SNTP_CLIENT, ST *)
FUNCTION_BLOCK SNTP_CLIENT
VAR_IN_OUT
	IP_C : IP_C; (* IP_Control Verwaltungsstruktur *)
	S_BUF : NETWORK_BUFFER;
	R_BUF : NETWORK_BUFFER;
END_VAR
VAR_INPUT
	IP4 : DWORD;
	ACTIVATE : BOOL;
END_VAR
VAR_OUTPUT
	ERROR : DWORD;
	DONE_P : BOOL;
	UDT : DT;
	XMS : INT;
END_VAR
VAR
	IP_FIFO : IP_FIFO;
	ip_state : BYTE;
	ip_id : BYTE;
	i : INT;
	last : DWORD;
	state : INT;
	tx : DWORD;
	activate_last : BOOL;
	ip4_stored : DWORD;

	(*LOG_MSG : LOG_MSG;
	_debug_enable : BOOL := TRUE;*)

END_VAR

(*
version 1.1		20. oct. 2009
programmer 		ks
tested by		ks

SNTP_CLIENT führt eine SNTP-Anfrage bei einem SNTP/NTP-Server um die aktuelle Uhrzeit zu erhalten
*)
(* Domain Name System (query) *)
tx := T_PLC_MS(); (* read system time *)

CASE state OF
00: (* auf positive Flanke SET warten *)
	DONE_P := FALSE;
	IF ACTIVATE AND NOT activate_last THEN
		ip4_stored := IP4; (* aktuelle IP4 speichern *)
		state := 10;
		ERROR := DWORD#0;
		ip_state := BYTE#1; (* Anmelden *)
		(*####################  DEBUG-MESSAGE  ###################################*)
		(*IF _debug_enable THEN
			LOG_CL.NEW_MSG := 'SNTP: S00 START';
			LOG_MSG();
		END_IF;*)
		(*########################################################################*)
	END_IF;

10: (* Bei IP_Control anmelden und auf freigabe warten *)
	IF ip_state = BYTE#3 THEN

		S_BUF.BUFFER[00] := BYTE#16#1B;
		FOR i := 1 TO 47 DO
			S_BUF.BUFFER[i] := BYTE#16#00;
		END_FOR;

		last := tx; (* aktuellen time wert sichern *)
		state := 30;

		(* IP Datenverkehr einrichten *)
		IP_C.C_PORT := WORD#123; (* Portnummer eintragen *)
		IP_C.C_IP := ip4_stored; (* IP eintragen *)
		IP_C.C_MODE := BYTE#1; (* Mode: UDP+AKTIV+PORT+IP *)
		IP_C.C_ENABLE := TRUE; (* Verbindungsaufbau freigeben *)
		IP_C.TIME_RESET := TRUE; (* Zeitueberwachung rücksetzen *)
		IP_C.R_OBSERVE := TRUE; (* Datenempfang ueberwachen *)
		S_BUF.SIZE := UINT#48; (* Sendelänge eintragen *)
		R_BUF.SIZE := UINT#0; (* Empfangslänge rücksetzen *)
    		(*####################  DEBUG-MESSAGE  ###################################*)
    		(*IF _debug_enable THEN
      			LOG_CL.NEW_MSG := 'SNTP: S10 SEND';
      			LOG_MSG();
    		END_IF;*)
    		(*########################################################################*)
	END_IF;

30:
	IF IP_C.ERROR <> DWORD#00 THEN
		ERROR := IP_C.ERROR;
		S_BUF.SIZE := UINT#0;
		R_BUF.SIZE := UINT#0;
		state := 0;
    		(*####################  DEBUG-MESSAGE  ###################################*)
    		(*IF _debug_enable THEN
      			LOG_CL.NEW_MSG := 'SNTP: S30 ERROR ~1';
      			LOG_CL.PRINTF[1] := DWORD_TO_STRING(ERROR);
      			LOG_MSG();
    		END_IF;*)
    		(*########################################################################*)

	ELSIF S_BUF.SIZE = UINT#0 AND R_BUF.SIZE >= UINT#48 THEN (* länge der empfangenen Daten prüfen *)

		(* Umrechnung SNTP Timestamp Base 1900-01-01 -> Unix 1970-01-01 = +2208988800 sekunden*)
		UDT := DWORD_TO_DT(DWORD_OF_BYTE(R_BUF.BUFFER[40],R_BUF.BUFFER[41],R_BUF.BUFFER[42],R_BUF.BUFFER[43]) - DWORD#2208988800);

		(* Original-Sekundenanteile sind als 32 Bit Fractal dargestellt *)
		(* ms nur mit veringerte Auflösung berechnen 1/65535 -> Highword verwenden *)
		XMS := DWORD_TO_INT(SHR(DINT_TO_DWORD(WORD_TO_DINT(WORD_OF_BYTE(R_BUF.BUFFER[44],R_BUF.BUFFER[45])) * DINT#1000),16));
		(* Zeitdifferenz (Laufzeitfehler) zwischen Send und Receive /2 teilen und addieren *)
		XMS := XMS + DWORD_TO_INT(SHR(tx - last,1));

		UDT := DWORD_TO_DT(DT_TO_DWORD(UDT) + (XMS / 1000)); (* sekundenanteile der Zeitdifferenz zu UDT aufrechnen *)
		XMS := XMS MOD 1000;  (* ms übernehmen *)
		state := 0;
		DONE_P := TRUE;
    		(*####################  DEBUG-MESSAGE  ###################################*)
    		(*IF _debug_enable THEN
        			LOG_CL.NEW_MSG := 'SNTP: S30 OK';
        			LOG_MSG();
    		END_IF;*)
    		(*########################################################################*)

	END_IF;

	IF state = 0 THEN
		IP_C.R_OBSERVE := FALSE; (* Datenempfang ueberwachen *)
		ip_state := BYTE#4;
	END_IF;

END_CASE;

activate_last := ACTIVATE; (* letzten Status sichern zur Flankenerkennung *)

(* IP_FIFO *)
IP_FIFO(FIFO:=IP_C.FIFO,STATE:=ip_state,ID:=ip_id);

(* revision history
ks	18. oct. 2008	rev 1.0
	original version

ks	20. oct. 2009	rev 1.1
	Networkbuffer und Buffer-funktionen auf Basis 0

*)

(***************************************************************************************)
(*               SNTP Datenstruktur
                                  1                   2                   3   
              0 1 2 3 4 5 6 7 8 9 0 1 2 3 4 5 6 7 8 9 0 1 2 3 4 5 6 7 8 9 0 1 
             +-+-+-+-+-+-+-+-+-+-+-+-+-+-+-+-+-+-+-+-+-+-+-+-+-+-+-+-+-+-+-+-+
Byte: 01-04  |LI | VN  |Mode |    Stratum    |     Poll      |   Precision   |
             +-+-+-+-+-+-+-+-+-+-+-+-+-+-+-+-+-+-+-+-+-+-+-+-+-+-+-+-+-+-+-+-+
Byte: 05-08  |                          Root  Delay (32 Bit)                 |
             +-+-+-+-+-+-+-+-+-+-+-+-+-+-+-+-+-+-+-+-+-+-+-+-+-+-+-+-+-+-+-+-+
Byte: 09-12  |                       Root  Dispersion (32 Bit)               |
             +-+-+-+-+-+-+-+-+-+-+-+-+-+-+-+-+-+-+-+-+-+-+-+-+-+-+-+-+-+-+-+-+
Byte: 13-16  |                     Reference Identifier (32 Bit)             |
             +-+-+-+-+-+-+-+-+-+-+-+-+-+-+-+-+-+-+-+-+-+-+-+-+-+-+-+-+-+-+-+-+
Byte: 17-24  |                    Reference Timestamp (64 Bit)               |
             +-+-+-+-+-+-+-+-+-+-+-+-+-+-+-+-+-+-+-+-+-+-+-+-+-+-+-+-+-+-+-+-+
Byte: 25-32  |                    Originate Timestamp (64 Bit)               |
             +-+-+-+-+-+-+-+-+-+-+-+-+-+-+-+-+-+-+-+-+-+-+-+-+-+-+-+-+-+-+-+-+
Byte: 33-40  |                     Receive Timestamp (64 Bit)                |
             +-+-+-+-+-+-+-+-+-+-+-+-+-+-+-+-+-+-+-+-+-+-+-+-+-+-+-+-+-+-+-+-+
Byte: 41-48  |                     Transmit Timestamp (64 Bit)               |
             +-+-+-+-+-+-+-+-+-+-+-+-+-+-+-+-+-+-+-+-+-+-+-+-+-+-+-+-+-+-+-+-+
Byte: 49-52  |                 Key Identifier (optional) (32 Bit)            |
             +-+-+-+-+-+-+-+-+-+-+-+-+-+-+-+-+-+-+-+-+-+-+-+-+-+-+-+-+-+-+-+-+
Byte: 53-68  |                 Message Digest (optional) (128 Bit)           |
             +-+-+-+-+-+-+-+-+-+-+-+-+-+-+-+-+-+-+-+-+-+-+-+-+-+-+-+-+-+-+-+-+

*)

(*
Worldwide NTP-Server


NIST-Zeitserver
• time-a.nist.gov
129.6.15.28 
NIST, Gaithersburg, Maryland 
• time-a.nist.gov
129.6.15.28 
NIST, Gaithersburg, Maryland 
• time-a.timefreq.bldrdoc.gov
132.163.4.101 (Stand: 1. Dezember 1999)
NIST, Boulder, Colorado 
• time-b.timefreq.bldrdoc.gov
132.163.4.102 (Stand: 1. Dezember 1999)
NIST, Boulder, Colorado 
• time-c.timefreq.bldrdoc.gov
132.163.4.103 (Stand: 1. Dezember 1999)
NIST, Boulder, Colorado 
• utcnist.colorado.edu
128.138.140.44
University of Colorado, Boulder 
• time.nist.gov
192.43.244.18
NCAR, Boulder, Colorado 
• time-nw.nist.gov
131.107.1.10
Microsoft, Redmond, Washington 
• nist1.dc.certifiedtime.com
216.200.93.8
Abovnet, North Virginia 
• nist1.datum.com
209.0.72.7
Datum, San Jose, Kalifornien 
• nist1.nyc.certifiedtime.com
208.184.49.129 
Abovnet, New York City 
• nist1.sjc.certifiedtime.com
207.126.103.202
Abovnet, San Jose, Kalifornien 

Zeitserver der ersten Ebene
Sortiert nach Standort: 
Nordamerika
• Palo Alto, Kalifornien: Systems Research Center, Compaq Computer Corp.
204.123.2.72: usno.pa-x.dec.com; CNAME: navobs1.pa-x.dec.com
Servicebereich: US-Zeitzonen PST (Pacific Standard Time) und MST (Mountain Standard Time) 
• Marina del Rey, Kalifornien: USC Information Sciences Institute
128.9.176.30: timekeeper.isi.edu
Servicebereich: CalRen2- und Los Nettos-Bereich  
• Washington, DC: U.S. Naval Observatory
192.5.41.41: tock.usno.navy.mil 
192.5.41.40: tick.usno.navy.mil
Servicebereich: NSFNET 
• Ottawa, Ontario, Kanada: National Research Council of Canada
time.chu.nrc.ca
Servicebereich: Kanada 
• Raleigh, North Carolina: North Carolina State University
152.1.58.124: terrapin.csc.ncsu.edu
Servicebereich: Südosten der USA 
• Cambridge, Massachusetts: MIT Information Systems
18.72.0.3: bitsy.mit.edu 
Servicebereich: NSFNET- und NEARnet-Bereich 
• Cambridge, Massachusetts: MIT
18.26.4.105: bonehed.lcs.mit.edu
Servicebereich: Osten der USA 
• Palo Alto, Kalifornien: Internet Software Consortium
192.5.5.250: clock.isc.org
Servicebereich: BARRnet, Alternet-West und CIX-West 
• Cambridge, Massachusetts: Open Software Foundation
130.105.4.59: clock.osf.org
Servicebereich: NSFNET- und NEARnet-Bereich 
• Palo Alto, Kalifornien: ViaNet Communications
209.81.9.7: clock.via.net 
• Cleveland, Ohio: Lewis Research Center (NASA)
128.156.1.43: lerc-dns.lerc.nasa.gov
Servicebereich: NSFNET und OARNET 
• Colorado Springs, Colorado: Schriever AFB
204.34.198.40: navobs1.usnogps.navy.mil; CNAME: tick.usnogps.navy.mil 
204.34.198.41: navobs1.usnogps.navy.mil; CNAME: tock.usnogps.navy.mil 
Servicebereich: US-Zeitzonen PST (Pacific Standard Time) und MST (Mountain Standard Time) 
• St. Louis, Missouri: Washington University
128.252.19.1: navobs1.usnogps.navy.mil; CNAME: tick.wustl.edu 
Servicebereich: US-Zeitzone CST (Central Standard Time) 
• Research Triangle Park, North Carolina: MCNC
192.101.21.1: ncnoc.ncren.net
Servicebereich: NC-REN-Bereich (North Carolina Research and Education Network) 
• Cupertino, Kalifornien: HP
192.6.38.127: ntp-cup.external.hp.com
Servicebereich: USA Westküste 
• Newark, Delaware: Conectiv Communications
138.39.7.20: ntp1.delmarva.com
Servicebereich: Cable & Wireless Network (früher MCInet) 
• University Park, Pennsylvania: Penn State University
128.118.46.3: otc1.psu.edu
Servicebereich: NSFNET, PREPNET und JvNCnet  

Europa
• Borowiec, Polen: Astrogeodynamical Observatory, Space Research Centre
150.254.183.15: vega.cbk.poznan.pl
Servicebereich: Polen und Europa 
• Stockholm, Schweden: Stupi AB
192.36.143.151: Time2.Stupi.SE
Servicebereich: Europa 
• Turin, Italien: IEN Galileo Ferraris
193.204.114.1: time.ien.it
Servicebereich: Italien und Europa 
• Zürich, Schweiz: Integrated Systems Laboratory , Eidgenössischen Technischen Hochschule Zürich 
129.132.2.21: swisstime.ethz.ch
Servicebereich: Schweiz und Europa 
• Turin, Italien: CSTV of National Research Council
150.145.33.1: tempo.cstv.to.cnr.it
Servicebereich: Italien und Europa 
• Erlangen, Deutschland: Universität Erlangen-Nürnberg
ntp0.fau.de; ntp1.fau.de; ntp2.fau.de; 
ntps1-0.uni-erlangen.de; ntps1-1.uni-erlangen.de; ntps1-2.uni-erlangen.de
Servicebereich: Deutschland und Europa 
• Berlin, Deutschland: Technische Universität Berlin
130.149.17.21: ntps1-0.cs.tu-berlin.de
130.149.17.8: ntps1-1.cs.tu-berlin.de
Servicebereich: Deutschland und Europa 
• Deutschland
131.173.17.7: ntps1-1.rz.Uni-Osnabrueck.DE
Servicebereich: Deutschland und Europa 
• Schweden
192.36.143.150: Time1.Stupi.SE
Servicebereich: SUnet und NORDUnet Schweden 

Fernost und pazifische Randgebiete
• Hong Kong: Chinesische Universität von Hong Kong. 
137.189.6.18: clock.cuhk.edu.hk
Servicebereich: Hong Kong (China) und Südostasien  
• Fukuoka, Japan: Universität Fukuoka
133.100.9.2: clock.nc.fukuoka-u.ac.jp
133.100.11.8: clock.tl.fukuoka-u.ac.jp
Servicebereich: Japan und pazifischer Raum  

Australien
• Melbourne, Australien: University of Melbourne
128.250.36.2: ntp.cs.mu.OZ.AU
Servicebereich: Australien und Neuseeland  

Zeitserver der zweiten Ebene
Nach geographischem Standort sortiert: 
Nordamerika
NTP-Zeitserver: • Quebec, Kanada: Canadian Meteorological Center
ntp1.cmc.ec.gc.ca; ntp2.cmc.ec.gc.ca 
Servicebereich: Ostkanada  
• Ontario, Kanada: National Research Council of Canada
time.chu.nrc.ca; time.nrc.ca
Servicebereich: Kanada 
• Saskatchewan, Kanada: University of Regina 
142.3.100.15: timelord.uregina.ca
Servicebereich: Kanada 
• Ontario, Kanada: University of Toronto
tick.utoronto.ca; tock.utoronto.ca
Servicebereich: Ostkanada  
• Mexiko: Audiotel-Büro 
ntp2a.audiotel.com.mx; ntp2c.audiotel.com.mx; ntp2b.audiotel.com.mx
Servicebereich: Avantel, MCINet und Mexiko 
• Santa Cruz, Kalifornien: Scruz-net, inc.
165.227.1.1: ns.scruz.net
Servicebereich: Westen der USA 
• San Diego, Kalifornien: UCSD Academic Computing Services/Network Operations
132.239.254.49: ntp.ucsd.edu
Servicebereich: CERFNET; NSFNET, SDSC-Bereich, und nahegelegene Bereiche 
• Quincy, Kalifornien 
ntp1.mainecoon.com; ntp2.mainecoon.com 
Servicebereich: Nordamerika 
• Newark, Delaware: University of Delaware
128.175.1.3: louie.udel.edu
Servicebereich: CAIRN, Abilene und vBNS  
• Atlanta, Georgia: CNSG
ntp.shorty.com
Servicebereich: Südwesten der USA  
• Kennesaw, Georgia: PeachNet 
rolex.peachnet.edu; timex.peachnet.edu
Servicebereich: PeachNet (Georgia) und Südwesten der USA  
• Urbana-Champaign, Illinois: University of Illinois
ntp-0.cso.uiuc.edu; ntp-1.cso.uiuc.edu; ntp-2.cso.uiuc.edu
Servicebereich: CICNET, Mittlerer Westen und NCSA-Bereich  
• Chicago, Illinois: Argonne National Laboratory 
ntp-1.mcs.anl.gov; ntp-2.mcs.anl.gov
Servicebereich: NSF/ANSNet, CICNet, NetIllinois und ESNet  
• West Lafayette, Indiana: Purdue University
gilbreth.ecn.purdue.edu; harbor.ecn.purdue.edu; molecule.ecn.purdue.edu 
Servicebereich: NSFNET- und CICNET-Bereich  
• Manhattan, Kansas: KansasNet OnLine Services
199.240.130.1: ntp1.kansas.net
199.240.130.12: ntp2.kansas.net
Servicebereich: Zentral-USA und Great Plains  
• Boston, Massachusetts: UMass-Boston CS dept.
158.121.104.4: timeserver.cs.umb.edu
Servicebereich: Neuengland  
• Minneapolis/St Paul, Minnesota: University of Minnesota
ns.nts.umn.edu; nss.nts.umn.edu
Servicebereich: CICNET-Bereich  
• Columbia, Missouri: University of Missouri-Columbia
128.206.206.12: everest.cclabs.missouri.edu
Servicebereich: MOREnet  
• Omaha, Nebraska: Radiks Internet Access
205.138.126.83: allison.radiks.net
Servicebereich: Mittlerer Westen, USA  
• Las Vegas, Nevada: University of Nevada System Computing Services
131.216.1.101: cuckoo.nevada.edu 
Servicebereich: NevadaNet, NSFNET und SDSC-Bereich  
• Las Vegas, Nevada: UNLV College of Engineering
tick.cs.unlv.edu; tock.cs.unlv.edu
Servicebereich: Sprintnet  
• New York City, New York: Columbia University
ntp.ctr.columbia.edu 
Servicebereich: Sprintlink und NYSERnet  
• Ithaca, New York: Cornell University 
192.35.82.50: ntp0.cornell.edu
Servicebereich: NSFNET und NYSER-Bereich  
• New York, New York: Morningside Campus, Columbia University
sundial.columbia.edu
Servicebereich: NYSERnet  
• New York City, New York: Columbia University Computer Science Department
timex.cs.columbia.edu 
Servicebereich: PSINET; NSFNET, und NYSER-Bereich  
• Norman, Oklahoma: University of Oklahoma
129.15.22.8: constellation.ecn.uoknor.edu 
Servicebereich: Midnet  
• Coos Bay, Oregon: Koala Computers
207.48.109.6: tick.koalas.com
Servicebereich: Nordwesten der USA  
• University Park, Pennsylvania: Penn State University
128.118.25.3: clock.psu.edu
Servicebereich: Internet2, vBNS, CERFnet(AT&T IP Services), PSC/NCNE und CASC 
• Pittsburgh, Pennsylvania: Pittsburgh Supercomputing Center
128.182.58.100: fuzz.psc.edu
Servicebereich: NSFNET und PSC-Bereich  
• Pittsburgh, Pennsylvania: Carnegie Mellon Electrical and Computer Engineering 
ntp-1.ece.cmu.edu; ntp-2.ece.cmu.edu 
Servicebereich: PREPNET und PSC-Bereich  
• Dallas, Texas: Cox School of Business, Southern Methodist University
129.119.80.126: ntp.cox.smu.edu 
Servicebereich: NSFNET und SESQUI-Bereich  
• Hughes Springs, Texas: First National Bank
209.144.20.76: ntp.fnbhs.com
Servicebereich: Nordosten Texas  
• Houston, Texas: Baylor College of Medicine
128.249.1.10: ntp.tmc.edu 
Servicebereich: NSFNET und SESQUI-Bereich  
• College Station, Texas: Texas A&M University
165.91.52.110: ntp5.tamu.edu
Servicebereich: NSFNET, SESQUI-Bereich, THEnet und TAMUSDSN 
• Plano, Texas: Greyware Automation Products
tick.greyware.com; tock.greyware.com
Servicebereich: Südzentral-USA  
• Blacksburg, Virginia: Virginia Tech Computing Center
ntp-1.vt.edu; ntp-2.vt.edu
Servicebereich: Südwesten der USA  
• Arlington, Virginia: Center for Seismic Studies
140.162.1.3: ntp.cmr.gov
Servicebereich: NSFNET und SURA-Bereich  
• Richland, Washington: Washington State University 
192.31.216.30: clock.tricity.wsu.edu
Servicebereich: NSFNET und NorthWestNet  
• Washington, USA: Mill Creek
time.ultimeth.net
Servicebereich: Nordwesten der USA  
• Wisconsin, USA: Computer Science Department, University of Wisconsin-Madison
ntp1.cs.wisc.edu; ntp2.cs.wisc.edu; ntp3.cs.wisc.edu
Servicebereich: USA und jeder andere  

Südamerika
• Buenos Aires, Argentinien: Network Access Point
200.49.40.1: CNAME: tick.nap.com.ar
200.49.32.1: CNAME: tock.nap.com.ar
Servicebereich: Argentinien 
• Buenos Aires, Argentinien: Sinectis S.A.
time.sinectis.com.ar 
Servicebereich: Argentinien 
• Brasilien: Brazilian Research Network
200.144.121.33: ntp.cais.rnp.br 
Servicebereich: Brasilien 
• Venezuela: VELUG, Grupo de Usuarios Linux de Venezuela
150.185.192.250: ntp.linux.org.ve
Servicebereich: Arica  

Europa
• Zürich, Schweiz: Eidgenössischen Technischen Hochschule Zürich
129.132.98.11: bernina.ethz.ch
Servicebereich: Schweiz und Europa  
• Standort: Kopenhagen, Dänemark, Europa 
clock.netcetera.dk; clock2.netcetera.dk 
Servicebereich: Dänemark, Skandinavien und Nordeuropa  
• Spanien: Altea 
slug.ctv.es
Servicebereich: Spanien  
• Pieksamaki, Finnland: Keski-Savon Oppimiskeskus
tick.keso.fi; tock.keso.fi
Servicebereich: Finnland  
• Meudon, Frankreich: Observatoire de Paris-Meudon 
ntp.obspm.fr 
Servicebereich: Frankreich und Europa  
• Lyon, Frankreich: CISM 
ntp.univ-lyon1.fr 
Servicebereich: Frankreich, Schweiz, Italien und Europa  
• Paris, Frankreich: VIA, Ecole Centrale
138.195.130.70: ntp.via.ecp.fr
Servicebereich: Frankreich und Europa  
• Budapest, Ungarn: KFKI Research Institute for Particle and Nuclear Physics
148.6.0.1: time.kfki.hu
Servicebereich: HUNGARNET  
• Italien: Net4u Srl, Vercelli, Italien
195.32.52.129: ntps.net4u.it
Servicebereich: Italien  
• Oslo, Norwegen: Universität Oslo
129.240.64.3: fartein.ifi.uio.no 
Servicebereich: NORDUnet  
• Oslo, Norwegen: Alcanet International
time.alcanet.no
Servicebereich: Europa 
• Krakau, Polen: Academic Computer Centre 
149.156.4.11: info.cyf-kr.edu.pl
Servicebereich: Polen und Europa  
• Lund, Schweden: Lund Institute of Technology
130.235.20.3: ntp.lth.se 
Servicebereich: Schweden und NORDUnet 
• Ljubljana, Slowenien: Institute of Biophysics, University of Ljubljana
biofiz.mf.uni-lj.si 193.2.69.11
Servicebereich: Slowenien und Europa  
• Ljubljana, Slowenien: Hydrometeorological Institute of Slovenia
hmljhp.rzs-hm.si
Servicebereich: Slowenien und Europa  
• Ljubljana, Slowenien: Academic and Research Network of Slovenia
ntp1.arnes.si; ntp2.arnes.si
Servicebereich: Slowenien und Europa  
• Ljubljana, Slowenien: J. Stefan Institute
time.ijs.si
Servicebereich: Slowenien und Europa  

Britische Inseln
• Dublin, Irland: School of Mathematics, Trinity College 
ntp.cs.tcd.ie; ntp.maths.tcd.ie; ntp.tcd.ie
Servicebereich: Irland und Großbritannien 
• Glasgow, Schottland: Strathclyde University 
ntp.cs.strath.ac.uk 
Servicebereich: Großbritannien, Europa und andere 
• Cambridge, Großbritannien
ntp0.uk.uu.net; ntp1.uk.uu.net; 
ntp2.uk.uu.net 
Servicebereich: UUNET (in Großbritannien früher auch als PIPEX bekannt) und Großbritannien.  
• Manchester, England: University of Manchester
ntp2a.mcc.ac.uk; ntp2b.mcc.ac.uk;
ntp2c.mcc.ac.uk; ntp2d.mcc.ac.uk 
Servicebereich: Großbritannien  
• Buckinghamshire, Großbritannien: Wibble U.K., Aylesbury
tick.tanac.net
Servicebereich: Großbritannien  

Asien
• Moskau, Russland: Landau Institute for Theoretical Physics
193.233.9.7: ntp.landau.ac.ru
Servicebereich: Russland  
• Russland: Pushchino (bei Moskau)
194.149.67.130: ntp.psn.ru
Servicebereich: Russland 
• Chernogolovka, Russland: Chernogolovka Scientific Center (bei Moskau)
193.233.46.10: sign.chg.ru
Servicebereich: Russland  

Fernost und pazifische Randgebiete
• Tokyo, Japan: Cyber Fleet, Inc.
203.139.30.195: ntp.cyber-fleet.net
Servicebereich: Japan und Ostasien  
• Seoul, Korea: Inet, Inc.
time.nuri.net
Servicebereich: Korea, Japan, Hong Kong und Ostasien  
• Hamilton, Neuseeland: Universität Waikato
truechimer.waikato.ac.nz; truechimer1.waikato.ac.nz; 
truechimer2.waikato.ac.nz; truechimer3.waikato.ac.nz
Servicebereich: Neuseeland  
• Singapur und Philippinen: 
ntp.shim.org 
Servicebereich: Singapur  

Afrika
• Lagos, Nigeria: Supernet300
ntp.supernet300.com
Servicebereich: Westafrika (hauptsächlich nigerischer NITEL-Backbone)  
• Pietermaritzburg, Südafrika: Natal University
143.128.82.200: ntp.cs.unp.ac.za
Servicebereich: Südafrika  

Australien
• Adelaide, Südaustralien: University of Adelaide
129.127.28.4: augean.eleceng.adelaide.edu.au
129.127.40.3: ntp.adelaide.edu.au
203.21.37.18: ntp.saard.net
Servicebereich: AARNet  
• Carlton, Victoria, Australien: eSec Limited
203.21.84.4: time.esec.com.au  

*)
END_FUNCTION_BLOCK

(* POU SNTP_SERVER, ST *)
FUNCTION_BLOCK SNTP_SERVER
VAR_IN_OUT
	IP_C : IP_C; (* IP_Control Verwaltungsstruktur *)
	S_BUF : NETWORK_BUFFER;
	R_BUF : NETWORK_BUFFER;
END_VAR
VAR_INPUT
	ENABLE : BOOL;
	STRATUM : BYTE := BYTE#1;
	UDT : DT;
	XMS : INT;
END_VAR
VAR
	IP_FIFO : IP_FIFO;
	ip_state : BYTE;
	ip_id : BYTE;
	i2 : INT;
	i : INT;
	timestamp_int : DWORD; (* Timestamp integer part *)
	timestamp_sek : DWORD; (* Timestamp fraction part (HIGH_WORD) *)
	ts_b : BYTE;
	state : INT;
	tx : UDINT;
	t : TON;

	(*LOG_MSG : LOG_MSG;
	_debug_enable : BOOL := TRUE;*)

END_VAR

(*
version 1.2		17. may. 2011
programmer 		ks
tested by			ks

SNTP_SERVER stellt Datum/Uhrzeit füR andere (S)NTP_CLIENTS zur Verfügung.
*)
(* Domain Name System (query) *)
tx := T_PLC_MS(); (* read system time *)

CASE state OF

00: (* Warten auf Freigabe *)
	IF ENABLE THEN
		state := 10;
		ip_state := BYTE#1; (* Anmelden *)
    		(*####################  DEBUG-MESSAGE  ###################################*)
    		(*IF _debug_enable THEN
      			LOG_CL.NEW_MSG := 'SNTP_SERVER: S00 START';
      			LOG_MSG();
    		END_IF;*)
    		(*########################################################################*)
	END_IF;

10: (* Bei IP_Control anmelden und auf freigabe warten *)
	IF ip_state = BYTE#3 THEN
		(* IP Datenverkehr einrichten *)
		IP_C.C_PORT := WORD#123; (* Portnummer eintragen *)
		IP_C.C_IP := DWORD#00; (* IP eintragen *)
		IP_C.C_MODE := BYTE#5; (* Mode: UDP+PASSIV+PORT *)
		IP_C.C_ENABLE := TRUE; (* Verbindungsaufbau freigeben *)
		IP_C.TIME_RESET := TRUE; (* Zeitueberwachung rücksetzen *)
		IP_C.R_OBSERVE := FALSE; (* Datenempfang ueberwachen *)
		S_BUF.SIZE := UINT#0; (* Sendelänge eintragen *)
		R_BUF.SIZE := UINT#0; (* Empfangslänge rücksetzen *)
		state := 20;
    		(*####################  DEBUG-MESSAGE  ###################################*)
    		(*IF _debug_enable THEN
      			LOG_CL.NEW_MSG := 'SNTP_SERVER: S10 INIT';
      			LOG_MSG();
    		END_IF;*)
    		(*########################################################################*)
	END_IF;
20:
	IF R_BUF.SIZE > UINT#0 THEN
		state := 20;
    		(*####################  DEBUG-MESSAGE  ###################################*)
    		(*IF _debug_enable THEN
      			LOG_CL.NEW_MSG := 'SNTP_SERVER: S20 REQUEST - Size: ~1';
      			LOG_CL.PRINTF[1] := UINT_TO_STRING(R_BUF.SIZE);
      			LOG_MSG();
    		END_IF;*)
    		(*########################################################################*)
		(* empfangenes Telegramm mit 00 auffüllen , wenn zu kurz ! und Sendebuffer mit 00 vorbelegen *)
		FOR i := 0 TO 47 DO
			IF INT_TO_UINT(i) > R_BUF.SIZE - 1 THEN
				R_BUF.BUFFER[i] := BYTE#00;
			END_IF;
			S_BUF.BUFFER[i] := BYTE#00;
		END_FOR;

		R_BUF.SIZE := UINT#0;

		(* Sendedaten aufbereiten *)
		S_BUF.BUFFER[0] := BYTE#2#11100; (* Flags: NO WARNING, NTP VERSION 3 , SERVER *)
		S_BUF.BUFFER[1] := STRATUM; (* Peer Clock Stratum: *)
		S_BUF.BUFFER[2] := BYTE#10; (* Peer Polling Intervall 2 hoch 10 = 1024 sek. *)
		S_BUF.BUFFER[3] := BYTE#16#FB; (* Peer Clock Precision: -5 = -31,25ms *)

		(* Umrechnung SNTP Timestamp Base 1900-01-01 = Unix 1970-01-01 + 2208988800 sekunden *)
		timestamp_int := DT_TO_DWORD(UDT) + DWORD#2208988800;

		(* Sekundenanteile sind als 32 Bit Fractal dargestellt *)
		(* nur mit veringerte Auflösung berechnen 1/65535 -> Highword verwenden *)
		(* Berechnung des Sekundenanteils: xms * 65535 / 1000 *)
		timestamp_sek := DINT_TO_DWORD(DWORD_TO_DINT(SHL(INT_TO_DWORD(XMS),16))/DINT#1000);

		ts_b := BYTE_OF_DWORD(timestamp_int,3); (* Timestamp Byte 3 *)
		S_BUF.BUFFER[16] := ts_b; (* Reference Timestamp *)
		S_BUF.BUFFER[32] := ts_b; (* Receive   Timestamp *)
		S_BUF.BUFFER[40] := ts_b; (* Transmit  Timestamp *)

		ts_b := BYTE_OF_DWORD(TIMESTAMP_INT,2); (* Timestamp Byte 2 *)
		S_BUF.BUFFER[17] := ts_b; (* Reference Timestamp *)
		S_BUF.BUFFER[33] := ts_b; (* Receive   Timestamp *)
		S_BUF.BUFFER[41] := ts_b; (* Transmit  Timestamp *)

		ts_b := BYTE_OF_DWORD(TIMESTAMP_INT,1); (* Timestamp Byte 1 *)
		S_BUF.BUFFER[18] := ts_b; (* Reference Timestamp *)
		S_BUF.BUFFER[34] := ts_b; (* Receive   Timestamp *)
		S_BUF.BUFFER[42] := ts_b; (* Transmit  Timestamp *)

		ts_b := BYTE_OF_DWORD(TIMESTAMP_INT,0); (* Timestamp Byte 0 *)
		S_BUF.BUFFER[19] := ts_b; (* Reference Timestamp *)
		S_BUF.BUFFER[35] := ts_b; (* Receive   Timestamp *)
		S_BUF.BUFFER[43] := ts_b; (* Transmit  Timestamp *)

		ts_b := BYTE_OF_DWORD(TIMESTAMP_SEK,1); (* Timestamp Byte 1 *)
		S_BUF.BUFFER[20] := ts_b; (* Reference Timestamp *)
		S_BUF.BUFFER[36] := ts_b; (* Receive   Timestamp *)
		S_BUF.BUFFER[44] := ts_b; (* Transmit  Timestamp *)

		ts_b := BYTE_OF_DWORD(timestamp_sek,0);	(* Timestamp Byte 0 *)
		S_BUF.BUFFER[21] := ts_b; (* Reference Timestamp *)
		S_BUF.BUFFER[37] := ts_b; (* Receive   Timestamp *)
		S_BUF.BUFFER[45] := ts_b; (* Transmit  Timestamp *)

		(* Byte 1-8 von Transmit-Time auf Originate-Time umkopieren *)
		i2 := 40;
		FOR i := 24 TO 31 DO
			S_BUF.BUFFER[i] := R_BUF.BUFFER[i2];
			i2 := i2 +1;
		END_FOR;

		S_BUF.SIZE := UINT#48; (* Daten senden *)

	ELSIF NOT ENABLE AND S_BUF.SIZE = UINT#0 THEN
		ip_state := BYTE#4; (* Abmelden *)
		state := 0;
	END_IF;

END_CASE;

t(IN:= IP_C.ERROR > DWORD#0, PT:=T#5s);
IF t.Q THEN
  IP_C.TIME_RESET := TRUE; (* Error Reset *)
END_IF;

(* IP_FIFO *)
IP_FIFO(FIFO:=IP_C.FIFO,STATE:=ip_state,ID:=ip_id);

(* revision history
ks	18. oct. 2008	rev 1.0
	original version

ks	20. oct. 2009	rev 1.1
	Networkbuffer und Buffer-funktionen auf Basis 0

ks	17. may. 2011	rev 1.2
	automatischer re-connect
*)


(*               SNTP(NTP) Datenstruktur
                                  1                   2                   3
              0 1 2 3 4 5 6 7 8 9 0 1 2 3 4 5 6 7 8 9 0 1 2 3 4 5 6 7 8 9 0 1
             +-+-+-+-+-+-+-+-+-+-+-+-+-+-+-+-+-+-+-+-+-+-+-+-+-+-+-+-+-+-+-+-+
Byte: 01-04  |LI | VN  |Mode |    Stratum    |     Poll      |   Precision   |
             +-+-+-+-+-+-+-+-+-+-+-+-+-+-+-+-+-+-+-+-+-+-+-+-+-+-+-+-+-+-+-+-+
Byte: 05-08  |                          Root  Delay (32 Bit)                 |
             +-+-+-+-+-+-+-+-+-+-+-+-+-+-+-+-+-+-+-+-+-+-+-+-+-+-+-+-+-+-+-+-+
Byte: 09-12  |                       Root  Dispersion (32 Bit)               |
             +-+-+-+-+-+-+-+-+-+-+-+-+-+-+-+-+-+-+-+-+-+-+-+-+-+-+-+-+-+-+-+-+
Byte: 13-16  |                     Reference Identifier (32 Bit)             |
             +-+-+-+-+-+-+-+-+-+-+-+-+-+-+-+-+-+-+-+-+-+-+-+-+-+-+-+-+-+-+-+-+
Byte: 17-24  |                    Reference Timestamp (64 Bit)               |
             +-+-+-+-+-+-+-+-+-+-+-+-+-+-+-+-+-+-+-+-+-+-+-+-+-+-+-+-+-+-+-+-+
Byte: 25-32  |                    Originate Timestamp (64 Bit)               |
             +-+-+-+-+-+-+-+-+-+-+-+-+-+-+-+-+-+-+-+-+-+-+-+-+-+-+-+-+-+-+-+-+
Byte: 33-40  |                     Receive Timestamp (64 Bit)                |
             +-+-+-+-+-+-+-+-+-+-+-+-+-+-+-+-+-+-+-+-+-+-+-+-+-+-+-+-+-+-+-+-+
Byte: 41-48  |                     Transmit Timestamp (64 Bit)               |
             +-+-+-+-+-+-+-+-+-+-+-+-+-+-+-+-+-+-+-+-+-+-+-+-+-+-+-+-+-+-+-+-+
Byte: 49-52  |                 Key Identifier (optional) (32 Bit)            |
             +-+-+-+-+-+-+-+-+-+-+-+-+-+-+-+-+-+-+-+-+-+-+-+-+-+-+-+-+-+-+-+-+
Byte: 53-68  |                 Message Digest (optional) (128 Bit)           |
             +-+-+-+-+-+-+-+-+-+-+-+-+-+-+-+-+-+-+-+-+-+-+-+-+-+-+-+-+-+-+-+-+
*)
END_FUNCTION_BLOCK

(* POU SYS_LOG, ST *)
FUNCTION_BLOCK SYS_LOG
VAR_IN_OUT
	IP_C : IP_C; (* IP_Control Verwaltungsstruktur *)
	S_BUF : NETWORK_BUFFER;
	R_BUF : NETWORK_BUFFER;
END_VAR
VAR_INPUT
	ACTIVATE : BOOL;
	LDT : DT;
	SERVER_IP4 : DWORD;
	PORT : WORD;
	FACILITY : BYTE;
	SEVERITY : BYTE;
	TAG : STRING(32);
	HOSTNAME : STRING;
	MESSAGE : STRING(STRING_LENGTH);
	OPTION : BYTE;
END_VAR
VAR_OUTPUT
	DONE_P : BOOL;
	ERROR : DWORD;
END_VAR
VAR
	ip_state : BYTE;
	ip_id : BYTE;
	IP_FIFO : IP_FIFO;
	activate_last : BOOL;
	state : INT;
	s1 : STRING(20);
	i : INT;

	(*LOG_MSG : LOG_MSG;
	_debug_enable : BOOL := TRUE;*)

END_VAR

(*
version 1.1		20. jun. 2009
programmer 		ks
tested by		ks

SYSLOG versendet Meldungen auf Basis des SYSLOG-Standards

*)
CASE state OF
00: (* auf positive Flanke SET warten *)
	IF ACTIVATE AND NOT ACTIVATE_LAST THEN
		state := 10;
		ERROR := DWORD#0;
		IP_STATE := BYTE#1; (* Anmelden *)
    		(*####################  DEBUG-MESSAGE  ###################################*)
    		(*IF _debug_enable THEN
      			LOG_CL.NEW_MSG := 'SYS_LOG: S00 START /IP_ID ~4';
      			LOG_CL.PRINTF[4]  := BYTE_TO_STRING(IP_ID);
      			LOG_MSG();
    		END_IF;*)
    		(*########################################################################*)
	END_IF;
	DONE_P := FALSE;

10: (* Bei IP_Control anmelden und auf freigabe warten *)
	IF IP_STATE = BYTE#3 THEN
		(* Sendedaten aufbereiten *)
		i := 0;
		IF (OPTION AND BYTE#0000_0001) = BYTE#00 THEN (* Option: no priority Code *)
			(* Priority:  '<xx>' als dezimalwert *)
			(* BYTE: xxxx x...  = Facility *)
			(*       .... .xxx  = Level *)
			s1 := REPLACE('<P>',BYTE_TO_STRING(SHL(FACILITY,3) OR (SEVERITY AND BYTE#0000_0111)),1,2);
		ELSE
			s1 := '';
		END_IF;

		IF (OPTION AND BYTE#0000_0010) = BYTE#00 THEN (* Option: No Use Syslog RFC Header *)
			(* 'month day hh:mm:ss ' *)
			s1 := CONCAT(s1,DT_TO_STRF(DTI:=LDT,MS:=0,FMT:='#E #W #N:#R:#T ',LANG:=1));
			_STRING_TO_BUFFER(STR:=s1,POS:=i,PT:=ADR(S_BUF.BUFFER),SIZE:=UINT#1024);
			i := i + LEN(s1);
			(* ' sourcename eintragen *)
			_STRING_TO_BUFFER(STR:=HOSTNAME,POS:=i,PT:=ADR(S_BUF.BUFFER),SIZE:=UINT#1024);
			i := i + LEN(HOSTNAME);
			S_BUF.BUFFER[i] := BYTE#32; (* leerzeichen einfuegen *)
			i := i + 1;
			(* ' tag eintragen *)
			_STRING_TO_BUFFER(STR:=TAG,POS:=i,PT:=ADR(S_BUF.BUFFER),SIZE:=UINT#1024);
			i := i + LEN(TAG);
			S_BUF.BUFFER[i] := BYTE#32; (* leerzeichen einfuegen *)
			i := i + 1;
		END_IF;

		(* ' message eintragen *)
		_STRING_TO_BUFFER(STR:=MESSAGE,POS:=i,PT:=ADR(S_BUF.BUFFER),SIZE:=UINT#1024);
		i := i + LEN(MESSAGE);

		IF (OPTION AND BYTE#0000_0100) > BYTE#00 THEN (* Option: Add a CR & LF to end of message *)
			S_BUF.BUFFER[i] := BYTE#13; (* Carriage Return einfuegen *)
			i := i + 1;
			S_BUF.BUFFER[i] := BYTE#10; (* Linefeed einfuegen *)
			i := i + 1;
		END_IF;

		state := 30;

		(* IP Datenverkehr einrichten *)
		IF (OPTION AND BYTE#2#0000_1000) > BYTE#00 THEN (* Option: TCP Mode *)
			IP_C.C_MODE := BYTE#0; (* Mode: TCP/AKTIV *)
		ELSE
			IP_C.C_MODE := BYTE#1; (* Mode: UDP/AKTIV *)
		END_IF;

		IF PORT = WORD#0 THEN (* keine Portnummer vorgegeben ? *)
			IF IP_C.C_MODE = BYTE#0 THEN (* Modus bestimmen  TCP oder UDP ? *)
				IP_C.C_PORT := WORD#1468; (* Standard Portnummer für Syslog over TCP *)
			ELSE
				IP_C.C_PORT := WORD#514; (* Standard Portnummer für Syslog over UDP *)
			END_IF;
		ELSE
			IP_C.C_PORT := PORT; (* uebergebene Portnummer eintragen *)
		END_IF;

		IP_C.C_IP := SERVER_IP4; (* IP eintragen *)
		IP_C.C_ENABLE := TRUE; (* Verbindungsaufbau freigeben *)
		IP_C.TIME_RESET := TRUE; (* Zeitueberwachung rücksetzen *)
		IP_C.R_OBSERVE := FALSE; (* Datenempfang ueberwachen *)
		S_BUF.SIZE := INT_TO_UINT(i); (* Sendelänge eintragen *)
		R_BUF.SIZE := UINT#0; (* Empfangslänge rücksetzen *)
    		(*####################  DEBUG-MESSAGE  ###################################*)
    		(*IF _debug_enable THEN
      			LOG_CL.NEW_MSG := 'SYS_LOG: S20 SEND /IP_ID ~4';
      			LOG_CL.PRINTF[4]  := BYTE_TO_STRING(IP_ID);
      			LOG_MSG();
    		END_IF;*)
    		(*########################################################################*)
	END_IF;

